// ---- BaseClasses/FB_CycleProfiler.TcPOU
// Core §8.11.4(b)/(f) — the cycle-time profile, fed by the step record the chain
// already keeps for §6.9: StepChanged() from _M_SetStep (with the step's time class,
// WORK by default), CycleComplete() at the finish step (§8.11.1 marker). Application
// steps add NOTHING except one enum on genuine wait steps. The step-chain / Unit
// base (M2) calls both automatically; until then a Unit wires the two calls once
// (Annex C §C.6). Fixed-size, no runtime allocation (Core §8.11.4(e)).
FUNCTION_BLOCK FB_CycleProfiler
VAR_OUTPUT
    Current        : ST_CycleProfile;   // cycle in progress (live waterfall)
    LastCycle      : ST_CycleProfile;   // last completed cycle — the HMI chart source
    StepStats      : ARRAY[1..PL_Fraktal.MAX_PROFILE_STEPS] OF ST_TimingRow;  // per-StepNo aggregates
    StatsTruncated : BOOL;
    // §8.11.1 throughput markers + §8.11.4 trend ring (the cycle-time ANALYSIS source:
    // per-cycle work/wait-class totals, charted by the HMI to explain increases)
    LastCycleTime  : TIME;
    MinCycleTime   : TIME;              // rolling minimum since reset (the demonstrated best)
    History        : ARRAY[1..PL_Fraktal.MAX_CYCLE_HISTORY] OF ST_CycleSummary;
    HistoryHead    : INT;               // newest entry (0 = none yet)
    // §8.11.4(d) — degradation is data: WorkTime drifting beyond Baseline*(1+BandPct)
    // pulses DegradedTrig for ONE call so the owner raises the maintenance event once.
    BaselineWorkMs : UDINT;             // 0 = degradation watch off (§3.8 config)
    DegradedBandPct: UDINT := 20;       // allowed drift above baseline, percent
    DegradedTrig   : BOOL;
    DegradedWorkMs : UDINT;             // the WorkTime that tripped the band (for the event text)
END_VAR
VAR
    _running      : BOOL;
    _openNo       : INT;
    _openName     : STRING(80);
    _openClass    : E_TimeClass;
    _openExpected : TIME;
    _openStartMs  : DWORD;
    _openStartDt  : DT;
    _openStartSynchronized : BOOL;
    _cycleStartMs : DWORD;
    _degraded     : BOOL;               // latched: one event per excursion, not per cycle
END_VAR

// no cyclic body — event-driven via StepChanged/CycleComplete

// fold the open step into the profile, the class split, and the aggregates
METHOD PRIVATE _M_CloseOpen
VAR_INPUT
    NowMs : DWORD;
END_VAR
VAR
    dur  : DWORD;
    i    : INT;
    slot : INT;
END_VAR
IF _openNo = 0 THEN
    RETURN;
END_IF
dur := NowMs - _openStartMs;                                // wrap-safe (TC3 §8.11)

// (1) ordered waterfall entry
IF Current.NSteps < PL_Fraktal.MAX_PROFILE_STEPS THEN
    Current.NSteps := Current.NSteps + 1;
    Current.Steps[Current.NSteps].StepNo   := _openNo;
    Current.Steps[Current.NSteps].StepName := _openName;
    Current.Steps[Current.NSteps].TimeClass:= _openClass;
    Current.Steps[Current.NSteps].Started  := _openStartDt;
    Current.Steps[Current.NSteps].StartedTimeSynchronized := _openStartSynchronized;
    Current.Steps[Current.NSteps].Duration := DWORD_TO_TIME(dur);
    Current.Steps[Current.NSteps].Expected := _openExpected;
ELSE
    Current.Truncated := TRUE;
END_IF

// (2) time-class split (§8.11.4(f)) — WorkTime/WaitTime derive from this at cycle close
Current.ByClass[TO_INT(_openClass)] := Current.ByClass[TO_INT(_openClass)] + DWORD_TO_TIME(dur);

// (3) per-StepNo aggregate (find-or-allocate; fixed array, Core §8.11.4(e))
slot := 0;
FOR i := 1 TO PL_Fraktal.MAX_PROFILE_STEPS DO
    IF (StepStats[i].Count > 0) AND (StepStats[i].Id = _openNo) THEN
        slot := i;
        EXIT;
    ELSIF (slot = 0) AND (StepStats[i].Count = 0) THEN
        slot := i;
    END_IF
END_FOR
IF slot = 0 THEN
    StatsTruncated := TRUE;
ELSE
    StepStats[slot].Id        := _openNo;
    StepStats[slot].Label     := _openName;
    StepStats[slot].TimeClass := _openClass;
    F_TimingUpdate(Row := StepStats[slot], DurMs := dur);
END_IF
END_METHOD

// §8.11.1 — discard the OPEN cycle without publishing it: a stop accepted at the
// between-cycles wait must not count a wait-only fragment as a production cycle
// (it would poison MinCycleTime and the trend). Aggregates keep completed cycles.
METHOD CycleAbandon : BOOL
_running := FALSE;
_openNo := 0;
CycleAbandon := TRUE;
END_METHOD

// close the open step and publish the cycle (call at the finish step, §8.11.1).
// Publishes WorkTime = ByClass[WORK] — the real cycle time (§8.11.4(f)).
METHOD CycleComplete : BOOL
VAR
    nowMs : DWORD;
END_VAR
IF NOT _running THEN
    CycleComplete := FALSE;
    RETURN;
END_IF
nowMs := TIME_TO_DWORD(TIME());
_M_CloseOpen(nowMs);
Current.Total    := DWORD_TO_TIME(nowMs - _cycleStartMs);   // wrap-safe (TC3 §8.11)
Current.WorkTime := Current.ByClass[TO_INT(E_TimeClass.WORK)];
Current.WaitTime := Current.Total - Current.WorkTime;
Current.CycleNo  := LastCycle.CycleNo + 1;
LastCycle := Current;

// §8.11.1 throughput markers
LastCycleTime := Current.Total;
IF (MinCycleTime = T#0S) OR (Current.Total < MinCycleTime) THEN
    MinCycleTime := Current.Total;
END_IF

// §8.11.4 trend ring — per-cycle class split for the HMI's cause analysis
HistoryHead := (HistoryHead MOD PL_Fraktal.MAX_CYCLE_HISTORY) + 1;
History[HistoryHead].CycleNo  := Current.CycleNo;
History[HistoryHead].Started  := Current.Started;
History[HistoryHead].StartedTimeSynchronized := Current.StartedTimeSynchronized;
History[HistoryHead].Total    := Current.Total;
History[HistoryHead].WorkTime := Current.WorkTime;
History[HistoryHead].WaitTime := Current.WaitTime;
History[HistoryHead].ByClass  := Current.ByClass;

// §8.11.4(d) — degradation watch on WORK time (waits are attributed, not drift).
// One-call trigger, latched per excursion; recovery below the band rearms it.
DegradedTrig := FALSE;
DegradedWorkMs := TIME_TO_DWORD(Current.WorkTime);
IF BaselineWorkMs > 0 THEN
    IF DegradedWorkMs * 100 > BaselineWorkMs * (100 + DegradedBandPct) THEN
        IF NOT _degraded THEN
            _degraded := TRUE;
            DegradedTrig := TRUE;
        END_IF
    ELSE
        _degraded := FALSE;
    END_IF
END_IF

_running := FALSE;
_openNo  := 0;
CycleComplete := TRUE;
END_METHOD

// Configure the recipe-owned WORK-time reference through the profiler owner.
// BaselineWorkMs is published read-only; TwinCAT therefore rejects assignment
// through a parent FB's published Profiler output. Zero disables the watch.
METHOD M_SetBaselineWork : BOOL
VAR_INPUT
    WorkMs : UDINT;
END_VAR
BaselineWorkMs := WorkMs;
DegradedTrig := FALSE;
_degraded := FALSE;
M_SetBaselineWork := TRUE;
END_METHOD

// deliberate, LOGGED action only (Core §8.11.2) — the caller raises the event
METHOD ResetStats : BOOL
VAR
    i     : INT;
    empty : ST_TimingRow;
    emptySummary : ST_CycleSummary;
END_VAR
FOR i := 1 TO PL_Fraktal.MAX_PROFILE_STEPS DO
    StepStats[i] := empty;
END_FOR
FOR i := 1 TO PL_Fraktal.MAX_CYCLE_HISTORY DO
    History[i] := emptySummary;
END_FOR
HistoryHead := 0;
LastCycleTime := T#0S;
MinCycleTime := T#0S;
_degraded := FALSE;
StatsTruncated := FALSE;
LastCycle.CycleNo := 0;
ResetStats := TRUE;
END_METHOD

// call on every step change — _M_SetStep already has StepNo/StepName (§6.5).
// TimeClass defaults to WORK; only genuine wait steps pass a wait class (§8.11.4(f)).
METHOD StepChanged : BOOL
VAR_INPUT
    StepNo   : INT;
    StepName : STRING(120);
    TimeClass    : E_TimeClass;
    Expected : TIME;                   // §8.11.4(c) — declared guard, drawn vs actual
END_VAR
VAR
    nowMs : DWORD;
    i     : INT;
END_VAR
IF _running AND (StepNo = _openNo) THEN
    _openClass := TimeClass;               // same step refreshed — class may be (re)declared
    _openExpected := Expected;
    StepChanged := TRUE;
    RETURN;
END_IF
nowMs := TIME_TO_DWORD(TIME());
IF NOT _running THEN
    _running := TRUE;                  // first step opens the cycle (§8.11.1 start marker)
    _cycleStartMs := nowMs;
    Current.Started   := F_Now();
    Current.StartedTimeSynchronized := F_TimeSynchronized();
    Current.NSteps    := 0;
    Current.Truncated := FALSE;
    FOR i := 0 TO 4 DO
        Current.ByClass[i] := T#0S;    // reset the class split for the new cycle
    END_FOR
ELSE
    _M_CloseOpen(nowMs);
END_IF
_openNo      := StepNo;
_openName    := StepName;
_openClass   := TimeClass;
_openExpected := Expected;
_openStartMs := nowMs;
_openStartDt := F_Now();
_openStartSynchronized := F_TimeSynchronized();
StepChanged := TRUE;
END_METHOD

END_FUNCTION_BLOCK

// ---- BaseClasses/FB_HostEventPublisher.TcPOU
// Core §11.6 — bounded per-Unit L3 event projection. Event production is local;
// transport is an optional injected sink and can never command the Unit.
FUNCTION_BLOCK FB_HostEventPublisher
VAR_OUTPUT
    Ring     : ARRAY[1..PL_Fraktal.MAX_HOST_EVENTS] OF ST_HostEvent;
    RingHead : INT;       // newest record, 0 when empty
    Count    : INT;       // valid records, saturates at the bound
    Capacity : INT := PL_Fraktal.MAX_HOST_EVENTS; // published bound; clients do not duplicate it
    Wrapped  : BOOL;      // oldest records have been overwritten
END_VAR
VAR
    {attribute 'OPC.UA.DA' := '0'}
    _sink : I_HostEventSink;
    _sequence : UDINT;
END_VAR

// event-driven; no cyclic body

METHOD Emit : BOOL
VAR_INPUT
    Kind          : E_HostEventKind;
    StationPath   : STRING(255);
    PartUid       : STRING(64);
    Subject       : STRING(80);
    Value         : STRING(80);
    Verdict       : E_Verdict;
    ReasonCode    : E_Reason;
END_VAR
VAR
    validKind : BOOL;
END_VAR
Emit := FALSE;
CASE Kind OF
    E_HostEventKind.PART_RECEIVED,
    E_HostEventKind.PROCESSING_STARTED,
    E_HostEventKind.PROCESSED,
    E_HostEventKind.PROCESSING_ABORTED,
    E_HostEventKind.CHANGEOVER_STARTED,
    E_HostEventKind.CHANGEOVER_DONE,
    E_HostEventKind.TOOL_CHANGED,
    E_HostEventKind.MATERIAL_CHANGED,
    E_HostEventKind.MODE_CHANGED,
    E_HostEventKind.NOK:
        validKind := TRUE;
ELSE
    validKind := FALSE;
END_CASE
IF NOT validKind OR (StationPath = '') THEN
    RETURN;
END_IF
_sequence := _sequence + 1;
RingHead := (RingHead MOD PL_Fraktal.MAX_HOST_EVENTS) + 1;
Ring[RingHead].Sequence := _sequence;
Ring[RingHead].Kind := Kind;
Ring[RingHead].StationPath := StationPath;
Ring[RingHead].PartUid := PartUid;
Ring[RingHead].Subject := Subject;
Ring[RingHead].Value := Value;
Ring[RingHead].Stamp := F_Now();
Ring[RingHead].TimeSynchronized := F_TimeSynchronized();
Ring[RingHead].Verdict := Verdict;
Ring[RingHead].ReasonCode := ReasonCode;
IF Count < PL_Fraktal.MAX_HOST_EVENTS THEN
    Count := Count + 1;
ELSE
    Wrapped := TRUE;
END_IF
IF _sink <> 0 THEN
    _sink.OnHostEvent(Ev := Ring[RingHead]);
END_IF
Emit := TRUE;
END_METHOD

METHOD SetSink : BOOL
VAR_INPUT
    Sink : I_HostEventSink;
END_VAR
_sink := Sink;
SetSink := TRUE;
END_METHOD

END_FUNCTION_BLOCK

// ---- Connectivity/FB_LineData.TcPOU
// Core §3.8e - data shared by every station on a line, held once. A line is NOT
// part of the Unit forest: it is no Unit, EM or CM, has no parent, and is never
// registered as anyone's child. The composition root declares it beside the roots
// (as it does a control domain, §9.8) and every root on the line references it
// with SetLine. A project registers its line values here (the ordinary
// M_RegisterConfig* calls, Kind := LINE_CFG, keys 'line.*'); each referencing
// root publishes them as its own line data and routes their writes here, so they
// are edited, audited and access-classed exactly like any other value, through
// the one mailbox. It extends FB_ModuleBase only because the typed value registry
// lives there (ModuleType NONE); commands are refused.
//
// The OWNER is the only editable copy; every accepted change raises Revision and
// the whole line is republished as Image. A MIRROR, on another controller or a
// root that is not the owner's, obtains the owner's Image through I_LineSource and
// applies a new revision whole or not at all; its values are read-only to every
// client. A mirror that stops updating keeps running on the revision it has and
// says so (Stale): a shift boundary one revision old is a reporting error, not a
// hazard, so staleness never blocks production on its own (§3.8e(d)).
FUNCTION_BLOCK FB_LineData EXTENDS FB_ModuleBase
VAR_INPUT
    ParCfg : ST_LineDataParCfg;
    ParCmd : ST_LineDataParCmd;
END_VAR
VAR_OUTPUT
    OutCmd : ST_LineDataOutCmd;
    OutImm : ST_LineStatus;       // §3.8e(d) - what this copy says about itself
    Image      : ST_LineImage;    // what a mirror reads, by symbol, over its source
END_VAR
VAR PERSISTENT
    _revision : UDINT;            // owner: current; mirror: last applied
    Calendar  : ST_ShiftCalendar; // §8.5.2 - line data like any other: edited at the owner
END_VAR
VAR
    {attribute 'OPC.UA.DA' := '0'}
    _source : I_LineSource;
    {attribute 'OPC.UA.DA' := '0'}
    _log : POINTER TO FB_AlarmLog;
    _role          : E_LineRole;
    _lastOkMs      : DWORD;
    _applied       : BOOL;        // not persistent: every boot re-applies once
    _imageBuilt    : BOOL;
    _imageRevision : UDINT;
    _syncing       : BOOL;
    _staleEvt      : INT;
    {attribute 'OPC.UA.DA' := '0'}
    _host          : PVOID;       // the root that ticks this line and lends its alarm log
    {attribute 'OPC.UA.DA' := '0'}
    _schedule : FB_ShiftSchedule;
    _dailyView : ST_ShiftCalendarV3;
    _incoming      : ST_LineImage; // mirror staging buffer - an instance member, never a local
END_VAR

Cyclic();

// OWNER takes no source. A MIRROR needs one, and StaleAfterMs is the window it
// declares for staying current (§3.8e(d)). Name is the line's own identity, never
// a path under a Unit.
METHOD Setup : BOOL
VAR_INPUT
    Name         : STRING(80);
    LineId       : STRING(40);
    Role         : E_LineRole;
    Source       : I_LineSource;
    StaleAfterMs : UDINT;
END_VAR
_M_SetName(Name);
Setup := FALSE;
IF (LineId = '') OR ((Role <> E_LineRole.OWNER) AND (Role <> E_LineRole.MIRROR)) THEN
    RETURN;
END_IF
IF (Role = E_LineRole.MIRROR) AND (Source = 0) THEN
    RETURN;                                // a mirror with nothing to mirror
END_IF
_role := Role;
_source := Source;
ParCfg.StaleAfterMs := StaleAfterMs;
OutImm.LineId := LineId;
OutImm.Role := Role;
IF (Role = E_LineRole.OWNER) AND (_revision = 0) THEN
    _revision := 1;                        // a published line is never at revision 0
END_IF
_lastOkMs := TIME_TO_DWORD(TIME());
Setup := _M_RegisterCalendar();
END_METHOD

// §8.5.2(a) - every line carries a shift calendar, registered identically on owner
// and mirror so a mirror can apply the owner's line whole.
METHOD PROTECTED _M_RegisterCalendar : BOOL
VAR
    n    : INT;
    ok   : BOOL;
    key  : STRING(160);
    item : STRING(255);
    label : STRING(160);
END_VAR
ok := M_RegisterConfigNumber(Key := 'line.shift.utcOffsetMin', Item := 'Calendar/UtcOffsetMin',
    LabelKey := 'std.config.shiftUtcOffset', Unit := E_EngUnit.MINUTE, Kind := E_ConfigKind.LINE_CFG,
    Storage := E_ConfigStorage.AS_DINT, pTarget := ADR(Calendar.UtcOffsetMin),
    Minimum := -720.0, Maximum := 840.0, RequiresReady := FALSE);
FOR n := 1 TO PL_Fraktal.MAX_SHIFTS DO
    key := CONCAT('line.shift.', CONCAT(TO_STRING(n), '.startMin'));
    item := CONCAT('Calendar/StartMin[', CONCAT(TO_STRING(n), ']'));
    // One label per shift: the four sit together in a root's line data group.
    label := CONCAT('std.config.shift.', CONCAT(TO_STRING(n), '.start'));
    ok := M_RegisterConfigNumber(Key := key, Item := item, LabelKey := label,
        Unit := E_EngUnit.MINUTE, Kind := E_ConfigKind.LINE_CFG, Storage := E_ConfigStorage.AS_DINT,
        pTarget := ADR(Calendar.StartMin[n]), Minimum := -1.0, Maximum := 1439.0,
        RequiresReady := FALSE) AND ok;
END_FOR
_M_RegisterCalendar := ok;
END_METHOD

// §3.8e(a) - called by FB_UnitBase.SetLine. The FIRST root to reference the line
// hosts it: it ticks the line once per scan and lends its alarm log for the
// staleness event. Every later root only references it; the host binding again
// stays the host. TRUE = you host it.
METHOD M_BindHost : BOOL
VAR_INPUT
    pHost     : PVOID;
    pAlarmLog : POINTER TO FB_AlarmLog;
END_VAR
M_BindHost := FALSE;
IF (pHost = 0) OR ((_host <> 0) AND (_host <> pHost)) THEN
    RETURN;
END_IF
_host := pHost;
_log := pAlarmLog;
M_BindHost := TRUE;
END_METHOD

// §3.8e - a referencing root publishes the line's values as ITS line data: under
// the root's scope, items prefixed 'Line/', keys 'line.*' (M_RegisterConfigWrite
// holds every line key to that prefix, so they cannot collide with the root's).
METHOD M_AppendLineConfig : BOOL
VAR_INPUT
    Pager : REFERENCE TO FB_ConfigPager;
    Scope : STRING(255);
END_VAR
_M_AppendCapabilities(Pager := Pager, Scope := Scope, ItemPrefix := 'Line/');
M_AppendLineConfig := TRUE;
END_METHOD

// §8.5.2 - minutes after LOCAL midnight for a UTC timestamp, with the line's offset.
METHOD M_MinuteOfDay : DINT
VAR_INPUT
    Now : DT;
END_VAR
VAR
    secOfDay : DINT;
END_VAR
secOfDay := UDINT_TO_DINT(DT_TO_UDINT(Now) MOD 86400) + Calendar.UtcOffsetMin * 60;
secOfDay := ((secOfDay MOD 86400) + 86400) MOD 86400;   // normalize a negative offset
M_MinuteOfDay := secOfDay / 60;
END_METHOD

// §8.5.2(a) - the used shift in force at a local minute: the latest start at or
// before it, and before the day's first start the day's LAST shift (a night shift
// wraps midnight). 0 when no shift is used. Complete by construction: no gaps.
METHOD M_CurrentShift : INT
VAR_INPUT
    MinuteOfDay : DINT;
END_VAR
VAR
    n           : INT;
    best        : INT;
    bestStart   : DINT;
    latest      : INT;
    latestStart : DINT;
END_VAR
best := 0;
bestStart := -1;
latest := 0;
latestStart := -1;
FOR n := 1 TO PL_Fraktal.MAX_SHIFTS DO
    IF (Calendar.StartMin[n] >= 0) AND (Calendar.StartMin[n] <= 1439) THEN
        IF (Calendar.StartMin[n] <= MinuteOfDay) AND (Calendar.StartMin[n] > bestStart) THEN
            best := n;
            bestStart := Calendar.StartMin[n];
        END_IF
        IF Calendar.StartMin[n] > latestStart THEN
            latest := n;
            latestStart := Calendar.StartMin[n];
        END_IF
    END_IF
END_FOR
IF best = 0 THEN
    best := latest;
END_IF
M_CurrentShift := best;
END_METHOD

METHOD PROTECTED OnCyclic : DINT
OnCyclic := SUPER^.OnCyclic();
CASE _role OF
    E_LineRole.OWNER:
        _M_BuildImage();
        OutImm.Owner := Status.Name;
        OutImm.Stale := FALSE;
    E_LineRole.MIRROR:
        _M_Mirror();
ELSE
    ;                                      // not set up: publishes nothing to mirror
END_CASE
OutImm.Revision := _revision;
END_METHOD

METHOD PROTECTED _M_Dispatch
_M_Fault(E_Reason.UNSUPPORTED_COMMAND, 'std.error.passiveInputHasNoCommand');
END_METHOD

METHOD PROTECTED _M_ConfigReadOnly : BOOL
_M_ConfigReadOnly := (_role = E_LineRole.MIRROR) AND NOT _syncing;
END_METHOD

// The owner's revision rises with every accepted change, so a mirror can tell a
// new line from the one it has. A mirror's own apply never counts.
METHOD M_ApplyConfigWrite : BOOL
VAR_INPUT
    Scope     : STRING(255);
    WriteKey  : STRING(160);
    Revision  : UDINT;
    TextValue : STRING(255);
    RootReady : BOOL;
END_VAR
M_ApplyConfigWrite := SUPER^.M_ApplyConfigWrite(Scope := Scope, WriteKey := WriteKey,
    Revision := Revision, TextValue := TextValue, RootReady := RootReady);
IF M_ApplyConfigWrite AND (_role = E_LineRole.OWNER) THEN
    _revision := _revision + 1;
END_IF
END_METHOD

// Republish the whole line when its revision moved (or on the first scan, after
// every value has been registered). Values change only through the write path.
METHOD PRIVATE _M_BuildImage
VAR
    i     : INT;
    count : INT;
END_VAR
IF _imageBuilt AND (_imageRevision = _revision) THEN
    RETURN;
END_IF
Image.LineId := OutImm.LineId;
Image.Owner := Status.Name;
Image.Revision := _revision;
count := 0;
FOR i := 1 TO _nConfigWrite DO
    IF (_pConfigWrite[i - 1].Kind = E_ConfigKind.LINE_CFG)
    AND (count < PL_Fraktal.MAX_LINE_RECORDS) THEN
        count := count + 1;
        Image.Records[count].WriteKey := _pConfigWrite[i - 1].Key;
        Image.Records[count].Revision := _pConfigWrite[i - 1].Revision;
        Image.Records[count].ValueText := _M_ConfigValueText(Idx := i);
    END_IF
END_FOR
Image.Count := count;
_imageRevision := _revision;
_imageBuilt := TRUE;
END_METHOD

METHOD PRIVATE _M_Mirror
VAR
    ok      : BOOL;
    nowMs   : DWORD;
    elapsed : DWORD;
END_VAR
ok := FALSE;
nowMs := TIME_TO_DWORD(TIME());
IF _source.M_Poll(Image := _incoming) THEN
    IF _incoming.LineId <> OutImm.LineId THEN
        OutImm.SourceError := 1;       // somebody else's line: never applied
    ELSIF _applied AND (_incoming.Revision = _revision) THEN
        ok := TRUE;                        // current
    ELSIF _M_ApplyIncoming() THEN
        _revision := _incoming.Revision;
        _applied := TRUE;
        Image := _incoming;
        OutImm.Owner := _incoming.Owner;
        ok := TRUE;
    ELSE
        OutImm.SourceError := 2;       // not applicable whole: nothing applied
    END_IF
ELSIF _source.M_Error() <> 0 THEN
    OutImm.SourceError := _source.M_Error();
END_IF
IF ok THEN
    _lastOkMs := nowMs;
    OutImm.SourceError := 0;
    OutImm.LastUpdate := F_Now();
    OutImm.TimeSynchronized := F_TimeSynchronized();
END_IF
// Unsigned subtraction: a wrapping millisecond counter never fakes an expiry.
elapsed := nowMs - _lastOkMs;
OutImm.Stale := elapsed > TO_DWORD(ParCfg.StaleAfterMs);
IF OutImm.Stale AND (_staleEvt = 0) AND (_log <> 0) THEN
    _staleEvt := _log^.Raise(Reason := E_Reason.NONE, Text := 'std.error.lineDataStale',
        Source := Status.Name, Severity := E_Severity.LOW, Category := E_Category.SYSTEM,
        ResetClass := E_ResetClass.AUTO_RESET);
ELSIF NOT OutImm.Stale AND (_staleEvt > 0) THEN
    IF _log <> 0 THEN
        _log^.Gone(Slot := _staleEvt);
    END_IF
    _staleEvt := 0;
END_IF
END_METHOD

// §3.8e(c) - whole or not at all. The image must carry exactly the line values
// this copy registered; every record is staged through its typed handler before
// any is applied, as a §3.8b set load is.
METHOD PRIVATE _M_ApplyIncoming : BOOL
VAR
    i     : INT;
    j     : INT;
    n     : INT;
    local : INT;
END_VAR
_M_ApplyIncoming := FALSE;
n := LIMIT(0, _incoming.Count, PL_Fraktal.MAX_LINE_RECORDS);
local := 0;
FOR i := 1 TO _nConfigWrite DO
    IF _pConfigWrite[i - 1].Kind = E_ConfigKind.LINE_CFG THEN
        local := local + 1;
    END_IF
END_FOR
IF (n <> local) OR (n <> _incoming.Count) THEN
    RETURN;                                // the two sides disagree on what the line is
END_IF
// Duplicate identities cannot substitute for a missing field.
FOR i := 1 TO n DO
    FOR j := i + 1 TO n DO
        IF _incoming.Records[i].WriteKey = _incoming.Records[j].WriteKey THEN RETURN; END_IF
    END_FOR
END_FOR
IF NOT M_BeginConfigBatch() THEN RETURN; END_IF
_syncing := TRUE;
FOR i := 1 TO n DO
    IF NOT M_StageConfigWrite(Scope := Status.Name, WriteKey := _incoming.Records[i].WriteKey,
            Revision := _incoming.Records[i].Revision,
            TextValue := _incoming.Records[i].ValueText, RootReady := TRUE) THEN
        M_EndConfigBatch();
        _syncing := FALSE;
        RETURN;
    END_IF
END_FOR
IF NOT M_ValidateConfigBatch() THEN
    M_EndConfigBatch(); _syncing := FALSE; RETURN;
END_IF
FOR i := 1 TO n DO
    M_ApplyConfigWrite(Scope := Status.Name, WriteKey := _incoming.Records[i].WriteKey,
        Revision := _incoming.Records[i].Revision,
        TextValue := _incoming.Records[i].ValueText, RootReady := TRUE);
END_FOR
M_CommitConfigBatch();
_syncing := FALSE;
_M_ApplyIncoming := TRUE;
END_METHOD

METHOD M_ShiftInterval : BOOL
VAR_INPUT
    Now : DT;
END_VAR
VAR_OUTPUT
    ShiftIndex : INT;
    StartAt : DT;
    EndAt : DT;
    Target : UDINT;
END_VAR
M_ShiftInterval := _schedule.M_MigrateV1(Source := Calendar, Target := _dailyView);
IF M_ShiftInterval THEN
    _schedule.M_Interval(Now := Now, Calendar := _dailyView,
        ShiftIndex => ShiftIndex, StartAt => StartAt, EndAt => EndAt, Target => Target);
END_IF
END_METHOD

METHOD M_BeginConfigBatch : BOOL
M_BeginConfigBatch := TRUE;
END_METHOD

METHOD M_ValidateConfigBatch : BOOL
M_ValidateConfigBatch := TRUE;
END_METHOD

METHOD M_EndConfigBatch
;
END_METHOD

METHOD M_CommitConfigBatch : BOOL
M_CommitConfigBatch := TRUE;
END_METHOD

END_FUNCTION_BLOCK

// ---- Connectivity/FB_ShiftSchedule.TcPOU
FUNCTION_BLOCK FB_ShiftSchedule

;

// Half-open weekly intervals, including Sunday-to-Monday wrap.
METHOD M_Validate : BOOL
VAR_IN_OUT
    Calendar : ST_ShiftCalendarV3;
END_VAR
VAR
    i, j, dayI, dayJ, delta : INT;
    startI, endI, startJ, endJ : DINT;
END_VAR
M_Validate := FALSE;
IF (Calendar.SchemaVersion <> 3) OR (Calendar.UtcOffsetMin < -840)
OR (Calendar.UtcOffsetMin > 840) THEN RETURN; END_IF
FOR i := 1 TO PL_Fraktal.MAX_WEEKLY_SHIFTS DO
    IF (Calendar.Rows[i].StartMin < -1) OR (Calendar.Rows[i].StartMin > 1439)
    OR (Calendar.Rows[i].DurationMin < 1) OR (Calendar.Rows[i].DurationMin > 1440)
    OR (Calendar.Rows[i].ActiveDays < 0) OR (Calendar.Rows[i].ActiveDays > 127)
    OR (Calendar.Rows[i].ProductionTarget < 0) THEN RETURN; END_IF
END_FOR
FOR i := 1 TO PL_Fraktal.MAX_WEEKLY_SHIFTS DO
    IF Calendar.Rows[i].StartMin >= 0 THEN
        FOR dayI := 0 TO 6 DO
            IF (TO_DWORD(Calendar.Rows[i].ActiveDays) AND SHL(DWORD#1, dayI)) <> 0 THEN
                startI := dayI * 1440 + Calendar.Rows[i].StartMin;
                endI := startI + Calendar.Rows[i].DurationMin;
                FOR j := i TO PL_Fraktal.MAX_WEEKLY_SHIFTS DO
                    IF Calendar.Rows[j].StartMin >= 0 THEN
                        FOR dayJ := 0 TO 6 DO
                            IF ((j <> i) OR (dayJ <> dayI))
                            AND ((TO_DWORD(Calendar.Rows[j].ActiveDays) AND SHL(DWORD#1, dayJ)) <> 0) THEN
                                FOR delta := -1 TO 1 DO
                                    startJ := dayJ * 1440 + Calendar.Rows[j].StartMin + delta * 10080;
                                    endJ := startJ + Calendar.Rows[j].DurationMin;
                                    IF (startI < endJ) AND (startJ < endI) THEN RETURN; END_IF
                                END_FOR
                            END_IF
                        END_FOR
                    END_IF
                END_FOR
            END_IF
        END_FOR
    END_IF
END_FOR
M_Validate := TRUE;
END_METHOD

// Called at interval entry/boundary, not on every production scan.
METHOD M_Interval : BOOL
VAR_INPUT
    Now : DT;
END_VAR
VAR_IN_OUT
    Calendar : ST_ShiftCalendarV3;
END_VAR
VAR_OUTPUT
    ShiftIndex : INT;
    StartAt : DT;
    EndAt : DT; // zero means no finite next boundary
    Target : UDINT;
END_VAR
VAR
    nowSec, localSec, weekStart, startSec, endSec, nextSec : LINT;
    dayNo : LINT;
    i, day, week : INT;
END_VAR
M_Interval := TRUE;
ShiftIndex := 0; StartAt := Now; EndAt := DT#1970-01-01-00:00:00; Target := 0;
nowSec := TO_LINT(DT_TO_UDINT(Now));
localSec := nowSec + Calendar.UtcOffsetMin * LINT#60;
dayNo := localSec / 86400;
IF localSec < 0 THEN dayNo := (localSec - 86399) / 86400; END_IF
weekStart := (dayNo - ((dayNo + 3 + 7) MOD 7)) * 86400;
nextSec := LINT#4294967296;
FOR i := 1 TO PL_Fraktal.MAX_WEEKLY_SHIFTS DO
    IF (Calendar.Rows[i].StartMin >= 0) AND (Calendar.Rows[i].ActiveDays > 0) THEN
        FOR day := 0 TO 6 DO
            IF (TO_DWORD(Calendar.Rows[i].ActiveDays) AND SHL(DWORD#1, day)) <> 0 THEN
                FOR week := -1 TO 1 DO
                    startSec := weekStart + week * LINT#604800 + day * LINT#86400
                        + Calendar.Rows[i].StartMin * LINT#60 - Calendar.UtcOffsetMin * LINT#60;
                    endSec := startSec + Calendar.Rows[i].DurationMin * LINT#60;
                    IF (startSec <= nowSec) AND (nowSec < endSec) THEN
                        ShiftIndex := i;
                        IF startSec >= 0 THEN StartAt := UDINT_TO_DT(TO_UDINT(startSec)); END_IF
                        IF endSec <= 4294967295 THEN EndAt := UDINT_TO_DT(TO_UDINT(endSec)); END_IF
                        Target := TO_UDINT(Calendar.Rows[i].ProductionTarget);
                    END_IF
                    IF (startSec > nowSec) AND (startSec < nextSec) THEN nextSec := startSec; END_IF
                END_FOR
            END_IF
        END_FOR
    END_IF
END_FOR
IF (ShiftIndex = 0) AND (nextSec <= 4294967295) THEN EndAt := UDINT_TO_DT(TO_UDINT(nextSec)); END_IF
END_METHOD

METHOD M_MigrateV1 : BOOL
VAR_IN_OUT
    Source : ST_ShiftCalendar;
    Target : ST_ShiftCalendarV3;
END_VAR
VAR
    i, j : INT;
    duration, distance : DINT;
END_VAR
M_MigrateV1 := FALSE;
Target.SchemaVersion := 3;
Target.UtcOffsetMin := Source.UtcOffsetMin;
FOR i := 1 TO PL_Fraktal.MAX_WEEKLY_SHIFTS DO
    Target.Rows[i].StartMin := -1;
    Target.Rows[i].DurationMin := 1440;
    Target.Rows[i].ActiveDays := 0;
    Target.Rows[i].ProductionTarget := 0;
END_FOR
FOR i := 1 TO PL_Fraktal.MAX_SHIFTS DO
    IF (Source.StartMin[i] < -1) OR (Source.StartMin[i] > 1439) THEN RETURN; END_IF
    IF Source.StartMin[i] >= 0 THEN
        duration := 1440;
        FOR j := 1 TO PL_Fraktal.MAX_SHIFTS DO
            IF (j <> i) AND (Source.StartMin[j] >= 0) THEN
                distance := (Source.StartMin[j] - Source.StartMin[i] + 1440) MOD 1440;
                IF distance = 0 THEN RETURN; END_IF
                IF distance < duration THEN duration := distance; END_IF
            END_IF
        END_FOR
        Target.Rows[i].StartMin := Source.StartMin[i];
        Target.Rows[i].DurationMin := duration;
        Target.Rows[i].ActiveDays := 127;
    END_IF
END_FOR
M_MigrateV1 := M_Validate(Calendar := Target);
END_METHOD

METHOD M_MigrateV2 : BOOL
VAR_IN_OUT
    Source : ST_ShiftCalendarV2;
    Target : ST_ShiftCalendarV3;
END_VAR
VAR
    i : INT;
END_VAR
M_MigrateV2 := FALSE;
IF Source.SchemaVersion <> 2 THEN RETURN; END_IF
Target.SchemaVersion := 3;
Target.UtcOffsetMin := Source.UtcOffsetMin;
FOR i := 1 TO PL_Fraktal.MAX_WEEKLY_SHIFTS DO
    Target.Rows[i].StartMin := -1;
    Target.Rows[i].DurationMin := 1440;
    Target.Rows[i].ActiveDays := 0;
    Target.Rows[i].ProductionTarget := 0;
END_FOR
FOR i := 1 TO PL_Fraktal.MAX_SHIFTS DO
    Target.Rows[i].StartMin := Source.Rows[i].StartMin;
    Target.Rows[i].DurationMin := Source.Rows[i].DurationMin;
    Target.Rows[i].ActiveDays := Source.Rows[i].ActiveDays;
END_FOR
M_MigrateV2 := M_Validate(Calendar := Target);
END_METHOD

END_FUNCTION_BLOCK

// ---- BaseClasses/FB_SystemHealthPublisher.TcPOU
// Core §2.7/§8.12 — one bounded, reusable health evaluator. Platform adapters
// supply measurements; this owner publishes live values and owns alarm edges.
FUNCTION_BLOCK FB_SystemHealthPublisher
VAR_OUTPUT
    Status : ST_SystemHealthStatus;
END_VAR
VAR
    {attribute 'OPC.UA.DA' := '0'}
    _log : POINTER TO FB_AlarmLog;
    _sourcePath : STRING(255);
    _taskOverrunSlot, _taskJitterSlot, _controllerSlot : INT;
    _cpuSlot, _memorySlot, _temperatureSlot, _fanSlot, _storageSlot : INT;
    _fieldbusSlot, _dcSlot, _timeSlot : INT;
END_VAR

;

METHOD Setup : BOOL
VAR_INPUT
    SourcePath : STRING(255);
    pAlarmLog  : POINTER TO FB_AlarmLog;
END_VAR
_sourcePath := SourcePath;
_log := pAlarmLog;
Status.SourcePath := SourcePath;
Setup := (_sourcePath <> '') AND (_log <> 0);
END_METHOD

METHOD Cyclic : BOOL
VAR_INPUT
    Input      : ST_SystemHealthInput;
    ParCfg     : ST_SystemHealthParCfg;
    Configured : BOOL;
END_VAR
VAR
    validCfg, taskOverrunBad, jitterBad, controllerBad : BOOL;
    cpuBad, memoryBad, temperatureBad, fanBad, storageBad : BOOL;
    fieldbusBad, dcBad, timeBad : BOOL;
END_VAR
validCfg := Configured AND (ParCfg.SchemaVersion = 1)
    AND (ParCfg.MaxTaskCycleUs > 0) AND (ParCfg.MaxTaskJitterUs > 0)
    AND (ParCfg.MaxCpuLoadPct > 0.0) AND (ParCfg.MaxCpuLoadPct <= 100.0)
    AND (ParCfg.MaxIpcTemperatureC > 0.0)
    AND (ParCfg.MinStorageHealthPct >= 0.0) AND (ParCfg.MinStorageHealthPct <= 100.0)
    AND (ParCfg.MaxTimeOffsetUs >= 0);

Status.Present := validCfg;
Status.SourcePath := _sourcePath;
Status.TaskAvailable := Input.TaskAvailable;
Status.TaskCycleUs := Input.TaskCycleUs;
Status.TaskJitterUs := Input.TaskJitterUs;
Status.TaskOverrun := Input.TaskOverrun;
Status.ControllerAvailable := Input.ControllerAvailable;
Status.CpuLoadPct := Input.CpuLoadPct;
Status.MemoryAvailableMb := Input.MemoryAvailableMb;
Status.IpcAvailable := Input.IpcAvailable;
Status.IpcTemperatureC := Input.IpcTemperatureC;
Status.FanHealthy := Input.FanHealthy;
Status.StorageHealthPct := Input.StorageHealthPct;
Status.FieldbusAvailable := Input.FieldbusAvailable;
Status.FieldbusMasterHealthy := Input.FieldbusMasterHealthy;
Status.LostFrameCount := Input.LostFrameCount;
Status.SlaveErrorCount := Input.SlaveErrorCount;
Status.DcAvailable := Input.DcAvailable;
Status.DcSynchronized := Input.DcSynchronized;
Status.TimeQuality := Input.TimeQuality;
Status.FanAvailable := Input.IpcAvailable AND Input.FanAvailable;
Status.StorageAvailable := Input.IpcAvailable AND Input.StorageAvailable;

taskOverrunBad := validCfg AND (NOT Input.TaskAvailable OR Input.TaskOverrun
    OR (Input.TaskCycleUs > ParCfg.MaxTaskCycleUs));
jitterBad := validCfg AND Input.TaskAvailable
    AND (Input.TaskJitterUs > ParCfg.MaxTaskJitterUs);
controllerBad := validCfg AND NOT Input.ControllerAvailable;
cpuBad := validCfg AND Input.ControllerAvailable
    AND (Input.CpuLoadPct > ParCfg.MaxCpuLoadPct);
memoryBad := validCfg AND Input.ControllerAvailable
    AND (Input.MemoryAvailableMb < ParCfg.MinMemoryAvailableMb);
temperatureBad := validCfg AND Input.IpcAvailable
    AND (Input.IpcTemperatureC > ParCfg.MaxIpcTemperatureC);
fanBad := validCfg AND Input.IpcAvailable AND Input.FanAvailable
    AND NOT Input.FanHealthy;
storageBad := validCfg AND Input.IpcAvailable AND Input.StorageAvailable
    AND (Input.StorageHealthPct < ParCfg.MinStorageHealthPct);
fieldbusBad := validCfg AND (Input.FieldbusAvailable
    AND (NOT Input.FieldbusMasterHealthy
        OR (Input.LostFrameCount > ParCfg.MaxLostFrames)
        OR (Input.SlaveErrorCount > ParCfg.MaxSlaveErrors))
    OR (ParCfg.RequireFieldbus AND NOT Input.FieldbusAvailable));
dcBad := validCfg AND ParCfg.RequireDcSync
    AND (NOT Input.DcAvailable OR NOT Input.DcSynchronized);
timeBad := validCfg AND ParCfg.RequireTimeSync
    AND (NOT Input.TimeQuality.Available OR NOT Input.TimeQuality.Synchronized
        OR (Input.TimeQuality.OffsetUs > ParCfg.MaxTimeOffsetUs)
        OR (Input.TimeQuality.OffsetUs < -ParCfg.MaxTimeOffsetUs));

_M_UpdateAlarm(Active := taskOverrunBad, Reason := E_Reason.TASK_OVERRUN,
    Text := 'std.system.taskOverrun', Slot := _taskOverrunSlot);
_M_UpdateAlarm(Active := jitterBad, Reason := E_Reason.TASK_JITTER_HIGH,
    Text := 'std.system.taskJitterHigh', Slot := _taskJitterSlot);
_M_UpdateAlarm(Active := controllerBad, Reason := E_Reason.CONTROLLER_METRICS_UNAVAILABLE,
    Text := 'std.system.controllerMetricsUnavailable', Slot := _controllerSlot);
_M_UpdateAlarm(Active := cpuBad, Reason := E_Reason.CPU_LOAD_HIGH,
    Text := 'std.system.cpuLoadHigh', Slot := _cpuSlot);
_M_UpdateAlarm(Active := memoryBad, Reason := E_Reason.MEMORY_LOW,
    Text := 'std.system.memoryLow', Slot := _memorySlot);
_M_UpdateAlarm(Active := temperatureBad, Reason := E_Reason.IPC_TEMP_HIGH,
    Text := 'std.system.ipcTemperatureHigh', Slot := _temperatureSlot);
_M_UpdateAlarm(Active := fanBad, Reason := E_Reason.IPC_FAN_FAULT,
    Text := 'std.system.ipcFanFault', Slot := _fanSlot);
_M_UpdateAlarm(Active := storageBad, Reason := E_Reason.STORAGE_HEALTH_LOW,
    Text := 'std.system.storageHealthLow', Slot := _storageSlot);
_M_UpdateAlarm(Active := fieldbusBad, Reason := E_Reason.FIELDBUS_MASTER_FAULT,
    Text := 'std.system.fieldbusMasterFault', Slot := _fieldbusSlot);
_M_UpdateAlarm(Active := dcBad, Reason := E_Reason.DC_SYNC_LOST,
    Text := 'std.system.dcSyncLost', Slot := _dcSlot);
_M_UpdateAlarm(Active := timeBad, Reason := E_Reason.TIME_SYNC_LOST,
    Text := 'std.system.timeSyncLost', Slot := _timeSlot);

Status.Healthy := validCfg AND NOT taskOverrunBad AND NOT jitterBad
    AND NOT controllerBad AND NOT cpuBad AND NOT memoryBad
    AND NOT temperatureBad AND NOT fanBad AND NOT storageBad
    AND NOT fieldbusBad AND NOT dcBad AND NOT timeBad;
Cyclic := validCfg;
END_METHOD

METHOD PRIVATE _M_UpdateAlarm
VAR_INPUT
    Active : BOOL;
    Reason : E_Reason;
    Text   : STRING(255);
END_VAR
VAR_IN_OUT
    Slot : INT;
END_VAR
IF Active THEN
    IF (Slot = 0) AND (_log <> 0) THEN
        Slot := _log^.Raise(Reason := Reason, Text := Text, Source := _sourcePath,
            Severity := E_Severity.LOW, Category := E_Category.SYSTEM,
            ResetClass := E_ResetClass.AUTO_RESET);
    END_IF
ELSE
    IF (Slot > 0) AND (_log <> 0) THEN
        _log^.Gone(Slot := Slot);
    END_IF
    Slot := 0;
END_IF
END_METHOD

END_FUNCTION_BLOCK

// ---- BaseClasses/FB_SignalTower.TcPOU
// Core §8.13 — single state/alarm/operator-action mapping plus bounded lamp test.
// Outputs are semantics only; the project Hardware Driver owns electrical I/O.
FUNCTION_BLOCK FB_SignalTower
VAR_OUTPUT
    Status : ST_SignalTowerOut;
END_VAR
VAR
    _testEdge : R_TRIG;
    _testTimer : TON;
    _testActive : BOOL;
END_VAR

;

METHOD Cyclic : BOOL
VAR_INPUT
    MachineState          : E_MachineState;
    AlarmActive           : BOOL;
    HighestSeverity       : E_Severity;
    OperatorActionRequired: BOOL;
    LampTestRequest       : BOOL;
    ParCfg                : ST_SignalTowerParCfg;
END_VAR
VAR
    duration : TIME;
END_VAR
duration := ParCfg.LampTestDuration;
IF (ParCfg.SchemaVersion <> 1) OR (duration <= T#0S) THEN
    duration := T#3S;
ELSIF duration > T#30S THEN
    duration := T#30S;
ELSE
    ;
END_IF
_testEdge(CLK := LampTestRequest);
IF _testEdge.Q THEN
    _testActive := TRUE;
    _testTimer(IN := FALSE);
END_IF
_testTimer(IN := _testActive, PT := duration);
IF _testTimer.Q THEN
    _testActive := FALSE;
    _testTimer(IN := FALSE);
END_IF

Status.Red := FALSE;
Status.Amber := FALSE;
Status.Green := FALSE;
Status.Blue := FALSE;
Status.White := FALSE;
Status.Horn := FALSE;
Status.TestActive := _testActive;
IF _testActive THEN
    Status.Red := TRUE;
    Status.Amber := TRUE;
    Status.Green := TRUE;
    Status.Blue := TRUE;
    Status.White := TRUE;
    Status.Horn := TRUE;
ELSE
    CASE MachineState OF
        E_MachineState.DOWN:
            Status.Red := TRUE;
        E_MachineState.BLOCKED, E_MachineState.STARVED, E_MachineState.CHANGEOVER:
            Status.Amber := TRUE;
        E_MachineState.PRODUCING:
            Status.Green := TRUE;
        E_MachineState.IDLE, E_MachineState.STOPPED:
            ;
        ELSE
            Status.Red := TRUE; // unknown state fails conspicuously
    END_CASE
    IF AlarmActive THEN
        CASE HighestSeverity OF
            E_Severity.HIGH:
                Status.Red := TRUE;
                Status.Green := FALSE;
                IF ParCfg.HornOnHigh THEN Status.Horn := TRUE; ELSE ; END_IF
            E_Severity.MED, E_Severity.LOW:
                IF NOT Status.Red THEN Status.Amber := TRUE; ELSE ; END_IF
            ELSE
                Status.Red := TRUE;
                Status.Green := FALSE;
        END_CASE
    ELSE
        ;
    END_IF
    IF OperatorActionRequired THEN
        IF ParCfg.OperatorUsesWhite THEN Status.White := TRUE; ELSE Status.Blue := TRUE; END_IF
    ELSE
        ;
    END_IF
END_IF
Cyclic := TRUE;
END_METHOD

END_FUNCTION_BLOCK

// ---- Platform/F_ManualEnable.TcPOU
// Core §9 — derive the manual-enable fact from the published safety devices.
// Pure, bounded, and fail-closed: no enabling device mirrored means NOT held,
// so a cell that never wired one cannot jog with its guards open by omission.
//
// Grepping for calls to this function lists every place in a codebase where
// motion is authorised by an enabling device. That auditability is the point of
// deriving it here rather than letting each station assemble the condition.
FUNCTION F_ManualEnable : ST_ManualEnableStatus
VAR_INPUT
    Safety : ST_SafetyStatus;
END_VAR
VAR
    i : INT;
END_VAR

// Fail-closed defaults (§5.6, O10): every early return leaves Held FALSE.
F_ManualEnable.Present    := FALSE;
F_ManualEnable.Held       := FALSE;
F_ManualEnable.DeviceName := '';

IF NOT Safety.Present THEN
    RETURN;                       // no safety facet at all -> nothing to permit with
END_IF

FOR i := 1 TO PL_Fraktal.MAX_SAFETY_DEVICES DO
    IF Safety.Devices[i].Present AND (Safety.Devices[i].Kind = E_SafetyDeviceKind.ENABLE_SWITCH) THEN
        F_ManualEnable.Present := TRUE;
        // Permitting is the POSITIVE state, exactly as an E-stop that is not
        // pressed publishes Ready/NOT DemandActive (§9). A released or
        // panic-squeezed enabling device demands the safe state like any other
        // device, so it fails every one of these tests.
        IF Safety.Devices[i].Ready
            AND NOT Safety.Devices[i].DemandActive
            AND NOT Safety.Devices[i].SafeStateActive
            AND NOT Safety.Devices[i].FaultActive
            AND Safety.Devices[i].FieldbusHealthy
            AND (Safety.Devices[i].State = E_SafetyState.READY)
            // A fault anywhere in the facet withdraws the permission even while
            // this device reads as held: a safety system reporting a fault is
            // not one to take permission from (O10). It must be tested HERE -
            // a check after the loop never ran, because a held device RETURNs.
            AND NOT Safety.FaultActive THEN
            F_ManualEnable.Held       := TRUE;
            F_ManualEnable.DeviceName := Safety.Devices[i].Name;
            RETURN;                   // first permitting device wins and names itself
        END_IF
    END_IF
END_FOR

END_FUNCTION

// ---- Connectivity/FB_LineDataV3.TcPOU
// Versioned weekly Line owner/mirror; inherited V1 image is retained for migration.
FUNCTION_BLOCK FB_LineDataV3 EXTENDS FB_LineData
VAR PERSISTENT
    CalendarV2 : ST_ShiftCalendarV2; // explicit V2 migration image, never reinterpreted
    CalendarV3 : ST_ShiftCalendarV3;
END_VAR
VAR
    {attribute 'OPC.UA.DA' := '0'}
    _weeklyConfig : ARRAY[1..21] OF ST_ConfigWriteDef;
    _candidate : ST_ShiftCalendarV3;
    _batch : BOOL;
END_VAR

Cyclic();

METHOD PROTECTED _M_RegisterCalendar : BOOL
VAR
    n : INT;
    ok : BOOL;
    found : UINT;
    key : STRING(160);
    item : STRING(255);
    label : STRING(160);
END_VAR
_M_RegisterCalendar := FALSE;
IF NOT _M_UseConfigRegistry(pRecords := ADR(_weeklyConfig), Capacity := 21) THEN RETURN; END_IF
IF CalendarV3.SchemaVersion = 0 THEN
    IF CalendarV2.SchemaVersion = 2 THEN
        ok := _schedule.M_MigrateV2(Source := CalendarV2, Target := _candidate);
    ELSIF CalendarV2.SchemaVersion = 0 THEN
        ok := _schedule.M_MigrateV1(Source := Calendar, Target := _candidate);
    ELSE
        // A present incompatible weekly image is not a missing image.
        ok := FALSE;
    END_IF
    IF ok THEN CalendarV3 := _candidate; END_IF
END_IF
IF NOT _schedule.M_Validate(Calendar := CalendarV3) THEN
    // Reject a real incompatible image visibly; keep the schedule empty.
    found := CalendarV3.SchemaVersion;
    IF found = 0 THEN found := 65535; END_IF
    M_RestoreStationCfg(pVersion := ADR(found), SchemaVersion := 3);
    CalendarV3.SchemaVersion := 3;
    CalendarV3.UtcOffsetMin := 0;
    FOR n := 1 TO PL_Fraktal.MAX_WEEKLY_SHIFTS DO
        CalendarV3.Rows[n].StartMin := -1;
        CalendarV3.Rows[n].DurationMin := 1440;
        CalendarV3.Rows[n].ActiveDays := 0;
        CalendarV3.Rows[n].ProductionTarget := 0;
    END_FOR
END_IF
ok := M_RegisterConfigNumber(Key := 'line.shift.utcOffsetMin', Item := 'CalendarV3/UtcOffsetMin',
    LabelKey := 'std.config.shiftUtcOffset', Unit := E_EngUnit.MINUTE, Kind := E_ConfigKind.LINE_CFG,
    Storage := E_ConfigStorage.AS_DINT, pTarget := ADR(CalendarV3.UtcOffsetMin),
    Minimum := -840.0, Maximum := 840.0, RequiresReady := FALSE);
M_SetConfigAccess(WriteKey := 'line.shift.utcOffsetMin', ClassId := '',
    MinReadLevel := E_AccessLevel.NONE, MinWriteLevel := E_AccessLevel.ENGINEER);
FOR n := 1 TO PL_Fraktal.MAX_WEEKLY_SHIFTS DO
    key := CONCAT('line.shift.', CONCAT(TO_STRING(n), '.startMin'));
    item := CONCAT('CalendarV3/Rows[', CONCAT(TO_STRING(n), ']/StartMin'));
    label := CONCAT('std.config.shift.', CONCAT(TO_STRING(n), '.start'));
    ok := M_RegisterConfigNumber(Key := key, Item := item, LabelKey := label,
        Unit := E_EngUnit.MINUTE, Kind := E_ConfigKind.LINE_CFG, Storage := E_ConfigStorage.AS_DINT,
        pTarget := ADR(CalendarV3.Rows[n].StartMin), Minimum := -1.0, Maximum := 1439.0,
        RequiresReady := FALSE) AND ok;
    M_SetConfigAccess(WriteKey := key, ClassId := '', MinReadLevel := E_AccessLevel.NONE,
        MinWriteLevel := E_AccessLevel.ENGINEER);
    key := CONCAT('line.shift.', CONCAT(TO_STRING(n), '.durationMin'));
    item := CONCAT('CalendarV3/Rows[', CONCAT(TO_STRING(n), ']/DurationMin'));
    label := CONCAT('std.config.shift.', CONCAT(TO_STRING(n), '.duration'));
    ok := M_RegisterConfigNumber(Key := key, Item := item, LabelKey := label,
        Unit := E_EngUnit.MINUTE, Kind := E_ConfigKind.LINE_CFG, Storage := E_ConfigStorage.AS_DINT,
        pTarget := ADR(CalendarV3.Rows[n].DurationMin), Minimum := 1.0, Maximum := 1440.0,
        RequiresReady := FALSE) AND ok;
    M_SetConfigAccess(WriteKey := key, ClassId := '', MinReadLevel := E_AccessLevel.NONE,
        MinWriteLevel := E_AccessLevel.ENGINEER);
    key := CONCAT('line.shift.', CONCAT(TO_STRING(n), '.activeDays'));
    item := CONCAT('CalendarV3/Rows[', CONCAT(TO_STRING(n), ']/ActiveDays'));
    label := CONCAT('std.config.shift.', CONCAT(TO_STRING(n), '.activeDays'));
    ok := M_RegisterConfigNumber(Key := key, Item := item, LabelKey := label,
        Unit := E_EngUnit.NONE, Kind := E_ConfigKind.LINE_CFG, Storage := E_ConfigStorage.AS_DINT,
        pTarget := ADR(CalendarV3.Rows[n].ActiveDays), Minimum := 0.0, Maximum := 127.0,
        RequiresReady := FALSE) AND ok;
    M_SetConfigAccess(WriteKey := key, ClassId := '', MinReadLevel := E_AccessLevel.NONE,
        MinWriteLevel := E_AccessLevel.ENGINEER);
    key := CONCAT('line.shift.', CONCAT(TO_STRING(n), '.productionTarget'));
    item := CONCAT('CalendarV3/Rows[', CONCAT(TO_STRING(n), ']/ProductionTarget'));
    label := CONCAT('std.config.shift.', CONCAT(TO_STRING(n), '.productionTarget'));
    ok := M_RegisterConfigNumber(Key := key, Item := item, LabelKey := label,
        Unit := E_EngUnit.PIECE, Kind := E_ConfigKind.LINE_CFG, Storage := E_ConfigStorage.AS_DINT,
        pTarget := ADR(CalendarV3.Rows[n].ProductionTarget), Minimum := 0.0, Maximum := 2147483647.0,
        RequiresReady := FALSE) AND ok;
    M_SetConfigAccess(WriteKey := key, ClassId := '', MinReadLevel := E_AccessLevel.NONE,
        MinWriteLevel := E_AccessLevel.ENGINEER);
END_FOR
_M_RegisterCalendar := ok;
END_METHOD

METHOD M_ShiftInterval : BOOL
VAR_INPUT
    Now : DT;
END_VAR
VAR_OUTPUT
    ShiftIndex : INT;
    StartAt : DT;
    EndAt : DT;
    Target : UDINT;
END_VAR
M_ShiftInterval := _schedule.M_Interval(Now := Now, Calendar := CalendarV3,
    ShiftIndex => ShiftIndex, StartAt => StartAt, EndAt => EndAt, Target => Target);
END_METHOD

METHOD M_StageConfigWrite : BOOL
VAR_INPUT
    Scope : STRING(255);
    WriteKey : STRING(160);
    Revision : UDINT;
    TextValue : STRING(255);
    RootReady : BOOL;
END_VAR
VAR
    i : INT;
    original : PVOID;
END_VAR
M_StageConfigWrite := FALSE;
IF NOT _batch THEN _candidate := CalendarV3; END_IF
IF NOT SUPER^.M_StageConfigWrite(Scope := Scope, WriteKey := WriteKey, Revision := Revision,
        TextValue := TextValue, RootReady := RootReady) THEN RETURN; END_IF
FOR i := 1 TO _nConfigWrite DO
    IF _pConfigWrite[i - 1].Key = WriteKey THEN
        original := _pConfigWrite[i - 1].pTarget;
        IF (original < ADR(CalendarV3)) OR (original >= ADR(CalendarV3) + SIZEOF(CalendarV3)) THEN RETURN; END_IF
        _pConfigWrite[i - 1].pTarget := ADR(_candidate) + (original - ADR(CalendarV3));
        M_StageConfigWrite := _M_StoreConfigValue(Idx := i, TextValue := TextValue, Commit := TRUE);
        _pConfigWrite[i - 1].pTarget := original;
        EXIT;
    END_IF
END_FOR
IF M_StageConfigWrite AND NOT _batch THEN
    M_StageConfigWrite := _schedule.M_Validate(Calendar := _candidate);
END_IF
END_METHOD

METHOD M_ApplyConfigWrite : BOOL
VAR_INPUT
    Scope : STRING(255);
    WriteKey : STRING(160);
    Revision : UDINT;
    TextValue : STRING(255);
    RootReady : BOOL;
END_VAR
M_ApplyConfigWrite := M_StageConfigWrite(Scope := Scope, WriteKey := WriteKey,
    Revision := Revision, TextValue := TextValue, RootReady := RootReady);
IF NOT M_ApplyConfigWrite THEN RETURN; END_IF
IF NOT _batch THEN
    CalendarV3 := _candidate;
    IF _role = E_LineRole.OWNER THEN _revision := _revision + 1; END_IF
END_IF
END_METHOD

METHOD M_BeginConfigBatch : BOOL
M_BeginConfigBatch := NOT _batch;
IF M_BeginConfigBatch THEN _candidate := CalendarV3; _batch := TRUE; END_IF
END_METHOD

METHOD M_ValidateConfigBatch : BOOL
M_ValidateConfigBatch := _batch AND _schedule.M_Validate(Calendar := _candidate);
END_METHOD

METHOD M_EndConfigBatch
_batch := FALSE;
END_METHOD

METHOD M_CommitConfigBatch : BOOL
M_CommitConfigBatch := M_ValidateConfigBatch();
IF M_CommitConfigBatch THEN
    CalendarV3 := _candidate;
    IF _role = E_LineRole.OWNER THEN _revision := _revision + 1; END_IF
END_IF
_batch := FALSE;
END_METHOD

END_FUNCTION_BLOCK

// ---- BaseClasses/FB_AsciiDeviceCM.TcPOU
// Core §3.15.1a — CM base for ASCII request/response devices over I_ByteChannel
// (vision sensors, code readers, gauges). One-outstanding-request state machine:
// SendRequest -> await terminated response -> _M_OnResponse hook; silence -> fault
// 10402. The framing and request rules are FB_AsciiLink's, shared with connectors
// (§1.1 O9); this CM adds what a CM owns: its faults and its bounded reconnect.
// Written ONCE against the neutral seam: porting = swap the channel (O4/O8).
FUNCTION_BLOCK ABSTRACT FB_AsciiDeviceCM EXTENDS FB_ControlModuleBase
VAR
    Host        : STRING(80);          // §3.8 config (per deployment)
    Port        : UINT;
    Terminator  : STRING(2) := '$R';   // CR default; device profile may override
    RespTimeout : TIME := T#2S;
    LinkState   : E_ByteChannelState;  // published (Annex D link facet)
    LastResponse: STRING(255);         // published (diagnosis)
END_VAR
VAR
    {attribute 'OPC.UA.DA' := '0'}
    _link      : FB_AsciiLink;
    _tRetry    : TON;
    _retryMs   : TIME := T#500MS;       // bounded backoff (doubles to 10s)
    _openTried : BOOL;                  // backoff spaces RE-tries; the first Open is immediate
END_VAR

;  // driven via Cyclic (base) -> OnCyclic below

// wire the transport + endpoint. Call from the profile's Setup after _M_SetName.
METHOD SetupDevice : BOOL
VAR_INPUT
    Chan : I_ByteChannel;
    DevHost : STRING(80);
    DevPort : UINT;
END_VAR
IF Chan = 0 OR DevHost = '' THEN
    _M_FaultN(PL_TcpDevReasons.DEV_CFG_INVALID, 'std.error.deviceConnectionNotConfigured');
    SetupDevice := FALSE;
    RETURN;
END_IF
_link.M_Bind(Chan := Chan);
Host := DevHost;
Port := DevPort;
SetupDevice := TRUE;
END_METHOD

// channel management + RX framing. Profiles override _M_OnResponse, not this.
METHOD PROTECTED OnCyclic : DINT
VAR
    evt : E_AsciiLinkEvent;
END_VAR
OnCyclic := SUPER^.OnCyclic();
_link.Terminator := Terminator;
_link.RespTimeout := RespTimeout;
evt := _link.M_Tick();
LinkState := _link.State;
IF LinkState = E_ByteChannelState.CLOSED THEN
    IF NOT _openTried THEN
        _openTried := TRUE;                        // first sight of CLOSED: connect NOW
        _link.M_Open(Host := Host, Port := Port);
        LinkState := _link.State;                  // a synchronous transport is OPEN this scan
    ELSE
        _tRetry(IN := TRUE, PT := _retryMs);       // failed before: bounded backoff (§3.15.2 spirit)
        IF _tRetry.Q THEN
            _tRetry(IN := FALSE);
            _link.M_Open(Host := Host, Port := Port);
            LinkState := _link.State;
            IF _retryMs < T#10S THEN
                _retryMs := _retryMs * 2;
            END_IF
        END_IF
    END_IF
ELSIF LinkState = E_ByteChannelState.OPEN THEN
    _openTried := FALSE;
    _retryMs := T#500MS;
END_IF
CASE evt OF
    E_AsciiLinkEvent.NONE:
        ;
    E_AsciiLinkEvent.RESPONSE:
        LastResponse := _link.LastResponse;
        _M_OnResponse(Response := _link.Response);
    E_AsciiLinkEvent.OVERFLOW:
        _M_FaultN(PL_TcpDevReasons.DEV_RX_OVERFLOW, 'std.error.deviceResponseOverflow');
    E_AsciiLinkEvent.CHANNEL_FAULT:
        _M_FaultN(PL_TcpDevReasons.DEV_CHANNEL_FAULT, 'std.error.transportChannelFault');
    E_AsciiLinkEvent.TIMEOUT:
        _M_FaultN(PL_TcpDevReasons.DEV_RESP_TIMEOUT, 'std.error.deviceResponseTimeout');
ELSE
    _M_FaultN(PL_TcpDevReasons.DEV_CHANNEL_FAULT, 'std.error.byteChannelStateInvalid');
END_CASE
END_METHOD

// issue one request (terminator appended). FALSE if not connected or one pending.
METHOD SendRequest : BOOL
VAR_INPUT
    Text : STRING(250);
END_VAR
IF NOT _link.M_IsOpen() THEN
    _M_FaultN(PL_TcpDevReasons.DEV_NOT_CONNECTED, 'std.error.deviceNotConnected');
    SendRequest := FALSE;
    RETURN;
END_IF
// A pending request is the one-outstanding contract, not a fault: refused quietly.
_link.Terminator := Terminator;
SendRequest := _link.M_Send(Text := Text);
END_METHOD

// profile hook: parse one terminated response. Raise DEV_PROTOCOL on garbage.
METHOD PROTECTED _M_OnResponse
VAR_INPUT
    Response : STRING(255);
END_VAR
;
END_METHOD

END_FUNCTION_BLOCK

// ---- Connectivity/FB_AsciiLink.TcPOU
// Core §3.15.1a - ASCII request/response over I_ByteChannel, written ONCE: terminator
// framing, the one-outstanding-request rule, the receive bound and the response
// timeout. It owns no open policy and raises nothing: each tick returns an event,
// and its owner decides what that means - FB_AsciiDeviceCM faults and reconnects
// on its own backoff; a connector on FB_DeviceConnectorBase leaves session,
// heartbeat and reconnect to that base (§3.15.2). One framing, two owners (§1.1 O9).
FUNCTION_BLOCK FB_AsciiLink
VAR_INPUT
    Terminator  : STRING(2) := '$R';   // CR default; a device profile may override
    RespTimeout : TIME := T#2S;
END_VAR
VAR_OUTPUT
    State        : E_ByteChannelState; // last observed transport state
    Pending      : BOOL;               // one request outstanding
    Response     : STRING(255);        // the response of the last RESPONSE event
    LastResponse : STRING(255);        // kept until the next response (diagnosis)
END_VAR
VAR
    {attribute 'OPC.UA.DA' := '0'}
    _chan  : I_ByteChannel;
    _rx    : STRING(255);
    _tResp : TON;
END_VAR

;  // driven through M_Tick by its owner

METHOD M_Bind : BOOL
VAR_INPUT
    Chan : I_ByteChannel;
END_VAR
_chan := Chan;
M_Bind := (Chan <> 0);
END_METHOD

// TRUE when the transport accepted the open (OPENING, or OPEN at once on a
// synchronous transport). Whether it then comes up is observed over scans.
METHOD M_Open : BOOL
VAR_INPUT
    Host : STRING(80);
    Port : UINT;
END_VAR
M_Open := FALSE;
IF _chan = 0 THEN
    RETURN;
END_IF
_chan.Open(Host := Host, Port := Port);
State := _chan.State();
M_Open := (State = E_ByteChannelState.OPEN) OR (State = E_ByteChannelState.OPENING);
END_METHOD

METHOD M_Close : BOOL
M_Close := FALSE;
Pending := FALSE;
_tResp(IN := FALSE);
_rx := '';
IF _chan = 0 THEN
    RETURN;
END_IF
M_Close := _chan.Close();
State := _chan.State();
END_METHOD

// LIVE transport state (the published State is one scan old).
METHOD M_IsOpen : BOOL
M_IsOpen := FALSE;
IF _chan = 0 THEN
    RETURN;
END_IF
M_IsOpen := (_chan.State() = E_ByteChannelState.OPEN);
END_METHOD

// Issue one request (terminator appended). FALSE when there is no channel, it is
// not OPEN, or a request is already outstanding - refused, never queued.
METHOD M_Send : BOOL
VAR_INPUT
    Text : STRING(250);
END_VAR
M_Send := FALSE;
// The null test is its own statement: TwinCAT does not short-circuit by default,
// so folding it into the next condition would still call State() on a null
// interface and fault the runtime.
IF _chan = 0 THEN
    RETURN;
END_IF
// LIVE state: the cached State is one scan old and would reject a request issued
// in the same scan the transport opened.
IF _chan.State() <> E_ByteChannelState.OPEN THEN
    RETURN;
END_IF
IF Pending THEN
    RETURN;
END_IF
Pending := _chan.Send(Text := CONCAT(Text, Terminator));
M_Send := Pending;
END_METHOD

// Run the transport one scan: drain, frame one response, watch the timeout.
METHOD M_Tick : E_AsciiLinkEvent
VAR
    pos : INT;
END_VAR
M_Tick := E_AsciiLinkEvent.NONE;
IF _chan = 0 THEN
    RETURN;
END_IF
_chan.Tick();
State := _chan.State();
CASE State OF
    E_ByteChannelState.CLOSED, E_ByteChannelState.OPENING:
        ;                                       // the owner decides when to open
    E_ByteChannelState.OPEN:
        _chan.Poll(Buffer := _rx);
        pos := FIND(_rx, Terminator);
        IF pos > 0 THEN
            Response := LEFT(_rx, pos - 1);
            _rx := DELETE(_rx, pos + LEN(Terminator) - 1, 1);
            Pending := FALSE;
            _tResp(IN := FALSE);
            LastResponse := Response;
            M_Tick := E_AsciiLinkEvent.RESPONSE;
            RETURN;
        ELSIF LEN(_rx) >= 250 THEN
            _rx := '';
            M_Tick := E_AsciiLinkEvent.OVERFLOW;
            RETURN;                             // first-out; the timeout still runs next scan
        END_IF
    E_ByteChannelState.FAULT:
        Pending := FALSE;
        _tResp(IN := FALSE);
        _chan.Close();
        M_Tick := E_AsciiLinkEvent.CHANNEL_FAULT;
        RETURN;
ELSE
    _chan.Close();
    M_Tick := E_AsciiLinkEvent.INVALID_STATE;
    RETURN;
END_CASE
_tResp(IN := Pending, PT := RespTimeout);
IF _tResp.Q THEN
    Pending := FALSE;
    _tResp(IN := FALSE);
    M_Tick := E_AsciiLinkEvent.TIMEOUT;
END_IF
END_METHOD

END_FUNCTION_BLOCK

// ---- Connectivity/F_AppendTopologyConfig.TcPOU
// Core §3.10.2/§10.5.1 — export the activation-static fieldbus identity (tags,
// addresses, wiring, hierarchy) into the config manifest. The live members
// (State/LinkOk/values/force/quality/fault) stay cyclically published; the
// static members carry OPC.UA.DA=0 in ST_BusNode/ST_IoChannel and reach the
// HMI only through this walk. Item fragments use the server's array naming
// (Nodes/Nodes[i]/..., Channels/Channels[j]/...) under the reserved scope
// '#Fieldbus' so a generic client can rebuild the exact browse paths.
// Only populated slots are exported — the empty tail of the bounded table
// costs nothing on the wire.
FUNCTION F_AppendTopologyConfig : BOOL
VAR_IN_OUT
    Topology : ST_FieldbusTopology;
    Pager    : FB_ConfigPager;
END_VAR
VAR
    i, j       : INT;
    nodeBase   : STRING(255);
    chanBase   : STRING(255);
    item       : STRING(255);
    forceableText : STRING(5);
END_VAR
VAR CONSTANT
    SCOPE_FIELDBUS : STRING(16) := '#Fieldbus';
END_VAR

F_AppendTopologyConfig := TRUE;
FOR i := 1 TO Topology.NodeCount DO
    IF (i < 1) OR (i > PL_Fraktal.MAX_BUS_NODES) THEN
        EXIT;                                       // defensive bound (§5.6)
    END_IF
    nodeBase := CONCAT('Nodes/Nodes[', CONCAT(TO_STRING(i), ']/'));
    Pager.M_Append(Scope := SCOPE_FIELDBUS,
        Item := CONCAT(nodeBase, 'Name'), ValueText := Topology.Nodes[i].Name);
    Pager.M_Append(Scope := SCOPE_FIELDBUS,
        Item := CONCAT(nodeBase, 'DescriptionKey'),
        ValueText := Topology.Nodes[i].DescriptionKey);
    Pager.M_Append(Scope := SCOPE_FIELDBUS,
        Item := CONCAT(nodeBase, 'TypeId'), ValueText := Topology.Nodes[i].TypeId);
    Pager.M_Append(Scope := SCOPE_FIELDBUS,
        Item := CONCAT(nodeBase, 'Address'), ValueText := Topology.Nodes[i].Address);
    Pager.M_AppendNumber(Scope := SCOPE_FIELDBUS,
        Item := CONCAT(nodeBase, 'ParentIdx'),
        Number := TO_DINT(Topology.Nodes[i].ParentIdx));
    Pager.M_AppendNumber(Scope := SCOPE_FIELDBUS,
        Item := CONCAT(nodeBase, 'ChannelCount'),
        Number := TO_DINT(Topology.Nodes[i].ChannelCount));
    FOR j := 1 TO Topology.Nodes[i].ChannelCount DO
        IF (j < 1) OR (j > PL_Fraktal.MAX_NODE_CHANNELS) THEN
            EXIT;                                   // defensive bound (§5.6)
        END_IF
        chanBase := CONCAT(nodeBase,
            CONCAT('Channels/Channels[', CONCAT(TO_STRING(j), ']/')));
        Pager.M_Append(Scope := SCOPE_FIELDBUS,
            Item := CONCAT(chanBase, 'Name'),
            ValueText := Topology.Nodes[i].Channels[j].Name);
        Pager.M_Append(Scope := SCOPE_FIELDBUS,
            Item := CONCAT(chanBase, 'DescriptionKey'),
            ValueText := Topology.Nodes[i].Channels[j].DescriptionKey);
        Pager.M_Append(Scope := SCOPE_FIELDBUS,
            Item := CONCAT(chanBase, 'Address'),
            ValueText := Topology.Nodes[i].Channels[j].Address);
        Pager.M_Append(Scope := SCOPE_FIELDBUS,
            Item := CONCAT(chanBase, 'Path'),
            ValueText := Topology.Nodes[i].Channels[j].Path);
        Pager.M_Append(Scope := SCOPE_FIELDBUS,
            Item := CONCAT(chanBase, 'ModulePath'),
            ValueText := Topology.Nodes[i].Channels[j].ModulePath);
        Pager.M_AppendNumber(Scope := SCOPE_FIELDBUS,
            Item := CONCAT(chanBase, 'Dir'),
            Number := TO_DINT(Topology.Nodes[i].Channels[j].Dir));
        Pager.M_AppendNumber(Scope := SCOPE_FIELDBUS,
            Item := CONCAT(chanBase, 'Kind'),
            Number := TO_DINT(Topology.Nodes[i].Channels[j].Kind));
        Pager.M_Append(Scope := SCOPE_FIELDBUS,
            Item := CONCAT(chanBase, 'Unit'),
            ValueText := Topology.Nodes[i].Channels[j].Unit);
        IF Topology.Nodes[i].Channels[j].Forceable THEN
            forceableText := 'TRUE';
        ELSE
            forceableText := 'FALSE';
        END_IF
        Pager.M_Append(Scope := SCOPE_FIELDBUS,
            Item := CONCAT(chanBase, 'Forceable'), ValueText := forceableText);
    END_FOR
END_FOR

END_FUNCTION

// ---- Connectivity/FB_DeviceConnectorBase.TcPOU
// Core §3.15 written once: session + heartbeat + LinkTimeout loss confirm +
// bounded exponential backoff reconnect + NO self-resume of dependents (that is
// the fronting CM's contract). A transport implements only _M_Open/_M_Close/
// _M_HbStart/_M_HbPoll. Row T7 of §5.7 is proven here once.
FUNCTION_BLOCK ABSTRACT FB_DeviceConnectorBase IMPLEMENTS I_DeviceConnector
VAR_INPUT
    HbPeriod    : TIME := T#1S;
    LinkTimeout : TIME := T#3S;
    BackoffMin  : TIME := T#500MS;
    BackoffMax  : TIME := T#10S;
    Reaction    : E_LinkReaction := E_LinkReaction.HOLD;   // consumed by the fronting CM
END_VAR
VAR
    _name      : STRING(80);
    _sessionUp : BOOL;
    _linked    : BOOL;
    _hbBusy    : BOOL;
    _lastSeen  : DT;
    _diag      : ST_Diagnostic;
    _tHb, _tLoss, _tBk : TON;
    _backoffMs : DINT;
END_VAR

Cyclic();

METHOD Connect : BOOL
Connect := _M_TryOpen();
END_METHOD

METHOD Cyclic : BOOL
IF NOT _sessionUp THEN
    // bounded exponential backoff (§3.15) — never a tight reconnect loop
    _tBk(IN := TRUE, PT := DINT_TO_TIME(_backoffMs));
    IF _tBk.Q THEN
        _tBk(IN := FALSE);
        IF NOT _M_TryOpen() THEN
            _backoffMs := MIN(_backoffMs * 2, TIME_TO_DINT(BackoffMax));
        END_IF
    END_IF
    Cyclic := TRUE;
    RETURN;
END_IF
// heartbeat: issue when due, poll while busy
IF NOT _hbBusy THEN
    _tHb(IN := TRUE, PT := HbPeriod);
    IF _tHb.Q THEN
        _tHb(IN := FALSE);
        _hbBusy := _M_HbStart();
    END_IF
ELSE
    CASE _M_HbPoll() OF
        E_HbResult.OK:
            _hbBusy := FALSE;
            _linked := TRUE;
            _lastSeen := F_Now();                 // §2.7
            _diag.ReasonCode := E_Reason.NONE;
            _diag.Description := '';
            _tLoss(IN := FALSE);                  // healthy beat resets loss confirm
        E_HbResult.FAIL:
            _hbBusy := FALSE;
            _M_Lost(E_Reason.DEVICE_PROTOCOL_ERROR, 'std.error.heartbeatBadReply');
            Cyclic := TRUE;
            RETURN;
        E_HbResult.PENDING:
            ;                                      // request still in flight
    ELSE
        _hbBusy := FALSE;
        _M_Lost(E_Reason.DEVICE_PROTOCOL_ERROR, 'std.error.heartbeatResultInvalid');
        Cyclic := TRUE;
        RETURN;
    END_CASE
END_IF
// confirm loss only after LinkTimeout without a healthy beat (§3.15.2)
_tLoss(IN := TRUE, PT := LinkTimeout);
IF _tLoss.Q THEN
    _M_Lost(E_Reason.LINK_TIMEOUT, 'std.error.heartbeatLapsed');
END_IF
Cyclic := TRUE;
END_METHOD

METHOD Disconnect : BOOL
_M_Close();
_sessionUp := FALSE;
_linked := FALSE;
Disconnect := TRUE;
END_METHOD

// I_Module command-release seam. The connector owns no PLCopen Execute latch;
// the fronting Control Module owns and releases the dependent device command.
// Disconnecting here would defeat the mandatory bounded reconnect policy (Core §3.15.2).
METHOD M_ReleaseCommand : BOOL
M_ReleaseCommand := TRUE;
END_METHOD

METHOD GetFaultSummary : ST_Diagnostic
GetFaultSummary := _diag;
END_METHOD

METHOD PrepareRecipe : BOOL
VAR_INPUT
    Model : ST_ModelId;
END_VAR
PrepareRecipe := TRUE;
END_METHOD

METHOD CommitRecipe
END_METHOD

METHOD AbortRecipe
END_METHOD

METHOD Setup : BOOL
VAR_INPUT
    Name : STRING(80);
END_VAR
_name := Name;
_backoffMs := TIME_TO_DINT(BackoffMin);
Setup := TRUE;
END_METHOD

METHOD PROTECTED ABSTRACT _M_Close : BOOL
END_METHOD

// PENDING while in flight; OK resets loss confirm; FAIL = protocol error
METHOD PROTECTED ABSTRACT _M_HbPoll : E_HbResult
END_METHOD

METHOD PROTECTED ABSTRACT _M_HbStart : BOOL
END_METHOD

// stamp the link first-out, drop the session; reconnection is backoff-bounded,
// resumption of dependent commands is NEVER automatic (§3.15/§9.3)
METHOD PROTECTED _M_Lost
VAR_INPUT
    Reason : E_Reason;
    Text   : STRING(255);
END_VAR
IF _diag.ReasonCode <> Reason THEN
    _diag.Since := F_Now();
    _diag.TimeSynchronized := F_TimeSynchronized();
END_IF
_diag.ReasonCode  := Reason;
_diag.Description := Text;
_diag.SourcePath  := _name;
_diag.Severity    := E_Severity.MED;
_diag.Category    := E_Category.SYSTEM;
F_RationalizeDiagnostic(Diag := _diag);
_linked := FALSE;
_hbBusy := FALSE;
_M_Close();
_sessionUp := FALSE;
END_METHOD

METHOD PROTECTED ABSTRACT _M_Open : BOOL
END_METHOD

METHOD PROTECTED _M_TryOpen : BOOL
IF _M_Open() THEN
    _sessionUp := TRUE;
    _backoffMs := TIME_TO_DINT(BackoffMin);
    _M_TryOpen := TRUE;
ELSE
    _M_TryOpen := FALSE;
END_IF
END_METHOD

PROPERTY FaultActive : BOOL
GET
FaultActive := (NOT _linked) AND (_diag.ReasonCode <> E_Reason.NONE);
END_GET
END_PROPERTY

// The connector reports link state/faults. HOLD is a configured loss reaction
// interpreted by the fronting Control Module; it is not connector lifecycle state.
PROPERTY HoldActive : BOOL
GET
HoldActive := FALSE;
END_GET
END_PROPERTY

PROPERTY LastSeen : DT
GET
LastSeen := _lastSeen;
END_GET
END_PROPERTY

PROPERTY Linked : BOOL
GET
Linked := _linked;
END_GET
END_PROPERTY

PROPERTY LinkReason : ST_Diagnostic
GET
LinkReason := _diag;
END_GET
END_PROPERTY

PROPERTY ModuleType : E_ModuleType
GET
ModuleType := E_ModuleType.CONTROL_MODULE;
END_GET
END_PROPERTY

PROPERTY Name : STRING(80)
GET
Name := _name;
END_GET
END_PROPERTY

PROPERTY State : E_ExecState
GET
State := SEL(FaultActive, E_ExecState.READY, E_ExecState.ERROR);
END_GET
END_PROPERTY

END_FUNCTION_BLOCK

// ---- Connectivity/FB_EcBusHealth.TcPOU
// Core §10.5.1 infrastructure service: read the REAL, live state of every
// EtherCAT slave directly from the fieldbus master (Tc2_EtherCAT) and publish it
// per node, so the HMI fieldbus tree mirrors XAE — independent of any Control-On
// or safety verdict. Auto-detects from hardware: the project supplies only the
// master AmsNetId ('' = local CPU) and how its topology node indices line up
// with the master's slave ordering (one offset), not per-node wiring.
//
// This is not a module tier and owns no process image. It calls
// FB_IoTopologyPublisher.M_SetNodeState for each mapped node.
FUNCTION_BLOCK FB_EcBusHealth
VAR
    {attribute 'OPC.UA.DA' := '0'}
    _pub : POINTER TO FB_IoTopologyPublisher;
    _netId : T_AmsNetId;          // EtherCAT MASTER device AmsNetId (see Setup)
    _firstSlaveNode : INT;        // topology node index of master slave #1
    _slaveCount : INT;            // how many slaves the master is asked about
    _masterNode : INT;            // topology node index of the master itself (0 = none)
    _attached : BOOL;

    // §10.5.1 — which topology node each MASTER SLAVE INDEX belongs to.
    // _slaveNode[i] = topology node of the master's slave i (0 = unmapped).
    //
    // The master enumerates only devices with an EtherCAT slave controller on
    // the process-data ring. A bus coupler (EK1200) and a passive end cap
    // (EL9011) are in the project tree and in the catalog, but the master never
    // lists them -- so "catalog position" and "master slave index" are NOT the
    // same sequence. Assuming they were shifted every state by one: the press
    // bench published the EL1809's state onto the coupler, the EL2809's onto the
    // EL1809, the EL6001's onto the EL2809, and left the real EL6001 and the end
    // cap reading OFFLINE while all three cards were in OP. A wrong state on the
    // right node is worse than no state: it is a plausible lie.
    //
    // Setup's FirstSlaveNode/SlaveCount form still works and fills this map
    // consecutively -- correct whenever every catalogued node really is a slave.
    _slaveNode : ARRAY[1..PL_Fraktal.MAX_BUS_NODES] OF INT;
    // Topology nodes that are catalogued but are NOT on the master's slave list
    // (couplers, end caps). Their state is inferred, never invented: they carry
    // the bus and are reachable exactly when the slaves behind them answer.
    _passiveNode : ARRAY[1..PL_Fraktal.MAX_BUS_NODES] OF INT;
    _passiveCount : INT;

    // Auto-detection of the EtherCAT master's AmsNetId (no project wiring): the
    // master's NetId is the local AMS NetId with the last two bytes replaced by
    // 2.1 (Beckhoff convention -- a PC 'a.b.c.d.1.1' has its EtherCAT master at
    // 'a.b.c.d.2.1'; the InfoSys FB_EcGetAllSlaveStates example uses exactly this
    // pairing). Overridable via Setup for non-standard configurations.
    {attribute 'OPC.UA.DA' := '0'}
    _fbLocalNetId : Tc2_Utilities.FB_GetLocalAmsNetId;
    _autoDetect : BOOL;           // TRUE = derive the master NetId at runtime
    {attribute 'OPC.UA.DA' := '0'}
    _netIdArr : T_AmsNetIdArr;    // scratch for the derived master NetId

    {attribute 'OPC.UA.DA' := '0'}
    _fbStates : Tc2_EtherCAT.FB_EcGetAllSlaveStates;
    // Bounded state buffer, one ST_EcSlaveState (deviceState + linkState) per
    // slave. Beckhoff declares pStateBuf as ARRAY[0..EC_MAX_SLAVES], so this
    // buffer is ZERO-BASED: slave i (1..n, master scan order) is _stateBuf[i-1].
    {attribute 'OPC.UA.DA' := '0'}
    _stateBuf : ARRAY[0..PL_Fraktal.MAX_BUS_NODES] OF Tc2_EtherCAT.ST_EcSlaveState;
    _step : INT;
    _tPoll : TON;
    // Demand gating (§10.5.1 diagnostic surface): only scan while a consumer
    // asks. _firstScanDone lets one scan run after Setup so M_BusOk() — which
    // feeds control logic, not a view — is never based on unread hardware.
    _scanRequested : BOOL;
    _firstScanDone : BOOL;

    // §8.12/§10.5 master health. Unlike the per-slave picture it is NOT
    // demand-gated: alarms and M_BusOk consume it every scan, so it is sampled
    // once a second whether or not anyone has the bus view open.
    {attribute 'OPC.UA.DA' := '0'}
    _fbDevState : Tc2_EtherCAT.FB_EcGetMasterDevState;
    {attribute 'OPC.UA.DA' := '0'}
    _fbFrames : Tc2_EtherCAT.FB_EcMasterFrameStatistic;
    {attribute 'OPC.UA.DA' := '0'}
    _fbCrc : Tc2_EtherCAT.FB_EcGetAllSlaveCrcErrors;
    {attribute 'OPC.UA.DA' := '0'}
    _crcBuf : ARRAY[0..PL_Fraktal.MAX_BUS_NODES] OF DWORD;
    _mPhase : INT;
    _mPoll : TON;
    _mSampled : BOOL;
    _mSampledAt : TIME;
    _mBaselined : BOOL;
    _mWindowStart : TIME;
    _mLostBase : UDINT;
    _mCrcBase : UDINT;
    _mLastWindowLost : UDINT;
    _mLastWindowCrc : UDINT;
END_VAR
VAR CONSTANT
    // Tc2_EtherCAT master device-state bits (F_ConvMasterDevStateToString): link
    // error 0x0001, I/O locked 0x0002, out of send resources 0x0010, watchdog
    // 0x0020, driver missing 0x0040, I/O reset 0x0080, a device in INIT/PRE-OP/
    // SAFE-OP 0x0100/0x0200/0x0400, a device in error 0x0800. The redundancy-only
    // bits 0x0004/0x0008 are not faults of a working line; DC is reported apart.
    MASTER_FAULT_BITS : WORD := 16#0FF3;
    MASTER_DC_NOT_IN_SYNC : WORD := 16#1000;
    MASTER_POLL : TIME := T#1S;
    MASTER_WINDOW : TIME := T#10S;
    MASTER_FRESH_FOR : TIME := T#3S;
END_VAR
VAR_OUTPUT
    // Diagnostics so a fieldbus read failure is visible instead of silently
    // showing every node as faulted. Published for the HMI/engineer.
    ReadOk : BOOL;                // last slave-state read succeeded
    LastErrorId : UDINT;          // ADS error of the last failed read (0 = none)
    SlavesReported : UINT;        // slaves the master reports (nSlaves output)
    NetIdMissing : BOOL;          // TRUE = InfoData.AmsNetId not linked (all zero)
    MasterNetId : T_AmsNetId;     // the resolved master NetId actually being used
    // TRUE = the master reports a different slave count than the project
    // topology declares (missing/extra hardware, or a config not activated).
    // §10.5.1: an unmatched mapping is a commissioning error, never guessed.
    CountMismatch : BOOL;

    // ---- Raw read-back diagnostics (commissioning aid) --------------------
    // The decoded E_NodeState alone cannot distinguish "the master said INIT"
    // from "we indexed or decoded it wrong". These publish the EXACT bytes the
    // master returned plus how each was interpreted, so a disagreement with XAE
    // is attributable to hardware, indexing, or decode without attaching a
    // debugger. Deliberately PUBLISHED (no 'OPC.UA.DA' := '0'): the point is
    // that an engineer can read them remotely over ADS/OPC UA.
    // Read them as: slot k holds slave k (master scan order), which this
    // library maps to topology node DiagNodeIndex[k].
    DiagRawDeviceState : ARRAY[1..8] OF BYTE;   // deviceState byte, as received
    DiagRawLinkState : ARRAY[1..8] OF BYTE;     // linkState byte, as received
    DiagDecodedState : ARRAY[1..8] OF INT;      // E_NodeState after decoding
    DiagNodeIndex : ARRAY[1..8] OF INT;         // topology node each slave maps to
    DiagBufferBytes : UDINT;                    // cbBufLen passed to the FB
    DiagEntrySize : UDINT;                      // SIZEOF(ST_EcSlaveState)
    DiagScanCount : UDINT;                      // completed reads (proves polling)
    DiagScanRequested : BOOL;                   // the §10.5.1 demand-gate state
    DiagFirstScanDone : BOOL;

    // ---- Master health (§8.12/§10.5): sampled every second, never gated ----
    MasterAvailable : BOOL;     // state, frame and CRC counters read within 3 s
    MasterDevState  : WORD;     // raw master device state (F_ConvMasterDevStateToString)
    MasterHealthy   : BOOL;     // available and no MASTER_FAULT_BITS set
    LostFrameCount  : UDINT;    // lost cyclic+queued frames: current or last 10 s window
    SlaveErrorCount : UDINT;    // summed slave CRC errors: current or last 10 s window
    DcSynchronized  : BOOL;     // available and DC not reported out of sync
    MasterErrorId   : UDINT;    // ADS error of the last failed master read (0 = none)
END_VAR

;

// Bind the publisher and describe how topology nodes map to master slaves.
// MasterNetIdArr = OPTIONAL override for the EtherCAT master's AmsNetId. Pass all
//   zeros (the normal case, e.g. an unassigned T_AmsNetIdArr) to AUTO-DETECT it at
//   runtime: the library reads the local AMS NetId and applies the Beckhoff master
//   convention (last two bytes -> 2.1), so no project wiring, no XAE checkbox and
//   no hand-typed address are needed. Supply a value only for a non-standard
//   configuration (e.g. a remote master, or several masters on one PC), typically
//   by linking that master's InfoData.AmsNetId.
// FirstSlaveNode = topology index of the first EtherCAT slave (the coupler);
// SlaveCount = number of consecutive topology nodes that are real slaves, in
// master scan order; MasterNodeIndex = topology index of the EtherCAT master
// itself, or 0 if not represented.
METHOD Setup : BOOL
VAR_INPUT
    Publisher : REFERENCE TO FB_IoTopologyPublisher;
    MasterNetIdArr : T_AmsNetIdArr;
    FirstSlaveNode : INT;
    SlaveCount : INT;
    MasterNodeIndex : INT;
END_VAR
VAR
    i : INT;
    anyNonZero : BOOL;
END_VAR
// All-zero (or omitted) = auto-detect; any explicit value is used verbatim.
anyNonZero := FALSE;
FOR i := 0 TO 5 DO
    IF MasterNetIdArr[i] <> 0 THEN
        anyNonZero := TRUE;
    END_IF
END_FOR

_attached := __ISVALIDREF(Publisher)
    AND (FirstSlaveNode >= 1)
    AND (SlaveCount >= 0)
    AND (SlaveCount <= PL_Fraktal.MAX_BUS_NODES);
IF _attached THEN
    _pub := ADR(Publisher);
    _autoDetect := NOT anyNonZero;
    IF anyNonZero THEN
        // Tc2_System helper: byte array -> 'a.b.c.d.e.f' string.
        _netId := Tc2_System.F_CreateAmsNetId(nIds := MasterNetIdArr);
        MasterNetId := _netId;
        NetIdMissing := FALSE;
        _step := 0;
    ELSE
        // Resolve the local NetId first (step -10), then start polling.
        _netId := '';
        MasterNetId := '';
        NetIdMissing := TRUE;   // cleared once auto-detection succeeds
        _step := -10;
    END_IF
    _firstSlaveNode := FirstSlaveNode;
    _slaveCount := SlaveCount;
    _masterNode := MasterNodeIndex;
    // Consecutive default: master slave i -> topology node FirstSlaveNode+i-1.
    // Correct only when EVERY catalogued node in that window is a real slave;
    // call M_MapSlaveNode to state the mapping explicitly when it is not.
    _passiveCount := 0;
    FOR i := 1 TO PL_Fraktal.MAX_BUS_NODES DO
        IF i <= _slaveCount THEN
            _slaveNode[i] := _firstSlaveNode + i - 1;
        ELSE
            _slaveNode[i] := 0;
        END_IF
        _passiveNode[i] := 0;
    END_FOR
END_IF
Setup := _attached;
END_METHOD

// §10.5.1 — state explicitly which topology node the master's slave [SlaveIndex]
// is, for a bus whose catalog is NOT one-to-one with the master's slave list.
//
// The master enumerates only devices with an EtherCAT slave controller on the
// process-data ring. A bus coupler or a passive end cap appears in the project
// tree and in the catalog, but never in that list, so the default consecutive
// mapping shifts every state onto its neighbour. Call this once per real slave,
// after Setup, and the shift is impossible:
//
//   _busHealth.Setup(..., FirstSlaveNode := 2, SlaveCount := 3, MasterNodeIndex := 1);
//   _busHealth.M_MapSlaveNode(SlaveIndex := 1, NodeIndex := 3);  // EL1809
//   _busHealth.M_MapSlaveNode(SlaveIndex := 2, NodeIndex := 4);  // EL2809
//   _busHealth.M_MapSlaveNode(SlaveIndex := 3, NodeIndex := 5);  // EL6001
//   _busHealth.M_MapPassiveNode(NodeIndex := 2);                 // EK1200 coupler
//   _busHealth.M_MapPassiveNode(NodeIndex := 6);                 // EL9011 end cap
METHOD M_MapSlaveNode : BOOL
VAR_INPUT
    SlaveIndex : INT;   // 1-based index in the master's slave list
    NodeIndex : INT;    // topology node this slave IS (0 clears the mapping)
END_VAR
M_MapSlaveNode := _attached
    AND (SlaveIndex >= 1) AND (SlaveIndex <= PL_Fraktal.MAX_BUS_NODES)
    AND (NodeIndex >= 0);
IF M_MapSlaveNode THEN
    _slaveNode[SlaveIndex] := NodeIndex;
END_IF
END_METHOD

// §10.5.1 — declare a catalogued node that carries the bus but is NOT a slave
// the master enumerates (bus coupler, end cap, power feed).
//
// Its state is INFERRED, never invented: the devices behind it can only answer
// if it is passing traffic, so it is OPERATIONAL exactly when the read
// succeeded and at least one real slave reported. Without this it would sit at
// OFFLINE forever on a perfectly healthy bus -- which is the same "plausible
// lie" the positional mapping produced, just in the other direction.
METHOD M_MapPassiveNode : BOOL
VAR_INPUT
    NodeIndex : INT;
END_VAR
M_MapPassiveNode := _attached
    AND (NodeIndex >= 1)
    AND (_passiveCount < PL_Fraktal.MAX_BUS_NODES);
IF M_MapPassiveNode THEN
    _passiveCount := _passiveCount + 1;
    _passiveNode[_passiveCount] := NodeIndex;
END_IF
END_METHOD

// Non-blocking cyclic refresh: (re)issue the slave-state read at a bounded rate,
// then publish each node's real state. On a read error every mapped node is
// marked OFFLINE (fail-visible: an unreachable master is not "operational").
METHOD M_Refresh
VAR
    i : INT;
    node : INT;
    mapped : E_NodeState;
    linkOk : BOOL;
    reported : INT;   // slaves the master actually returned this read
END_VAR
IF NOT _attached THEN
    RETURN;
END_IF

// Mirror the gate state every cycle so "why is it not updating?" is answerable
// from published data alone: from the outside a PARKED scanner and a STUCK one
// look identical.
DiagScanRequested := _scanRequested;
DiagFirstScanDone := _firstScanDone;

// Master health first: it is consumed by alarms and M_BusOk, never parked.
_M_SampleMaster();

// §10.5.1 is a DIAGNOSTIC surface: the bus picture is only consumed while the
// fieldbus view is open. Polling the master every 250 ms regardless costs ADS
// bandwidth and PLC time for data nobody is reading, so the read is demand-gated
// (M_RequestScan, set by the HMI opening the view / a mailbox request). While no
// consumer is active the state machine idles and the last published states are
// held — they are not falsified, just not refreshed.
// Exception: the FIRST scan after Setup always runs, so M_BusOk() (a control
// input, not a view) has real data without anyone opening the HMI.
IF NOT _scanRequested AND _firstScanDone THEN
    _tPoll(IN := FALSE);
    RETURN;
END_IF

// Drive the async read. Re-trigger on a slow poll so a stuck call cannot pin the
// task; FB_EcGetAllSlaveStates is edge-triggered by bExecute. The slave count is
// implied by cbBufLen (nSlave * SIZEOF(ST_EcSlaveState)); there is no count input.
CASE _step OF
    -10:
        // Auto-detect: ask the router for this PC's AmsNetId.
        _fbLocalNetId(bExecute := FALSE);
        _fbLocalNetId(bExecute := TRUE);
        _step := -5;
    -5:
        _fbLocalNetId(bExecute := FALSE);
        IF NOT _fbLocalNetId.bBusy THEN
            IF _fbLocalNetId.bError THEN
                // Cannot resolve: stay fail-visible and retry on the next poll.
                ReadOk := FALSE;
                LastErrorId := _fbLocalNetId.nErrId;
                NetIdMissing := TRUE;
                _M_PublishAllOffline();
                _step := -10;
            ELSE
                // Beckhoff convention: the EtherCAT master of a PC 'a.b.c.d.1.1'
                // is 'a.b.c.d.2.1'. Keep the first four bytes, force 2.1.
                _netIdArr := _fbLocalNetId.AddrBytes;
                _netIdArr[4] := 2;
                _netIdArr[5] := 1;
                _netId := Tc2_System.F_CreateAmsNetId(nIds := _netIdArr);
                MasterNetId := _netId;
                NetIdMissing := FALSE;
                _step := 0;
            END_IF
        END_IF
    0:
        _fbStates(bExecute := FALSE);
        _fbStates(sNetId := _netId,
            pStateBuf := ADR(_stateBuf),
            cbBufLen := TO_UDINT(_slaveCount) * SIZEOF(Tc2_EtherCAT.ST_EcSlaveState),
            bExecute := (_slaveCount > 0));
        _step := 10;
    10:
        _fbStates(bExecute := FALSE);
        IF NOT _fbStates.bBusy THEN
            // Publish diagnostics every cycle so a failing read is visible.
            ReadOk := NOT _fbStates.bError;
            LastErrorId := _fbStates.nErrId;
            SlavesReported := _fbStates.nSlaves;
            IF NOT _fbStates.bError THEN
                // Only the first nSlaves buffer entries were written by the
                // master; the rest keep their previous/zero content. Decoding a
                // zeroed entry yields linkState 0, which reads as "link OK" — a
                // FAIL-OPEN that showed absent slaves as healthy. Publish only
                // what the master actually reported and mark the surplus
                // OFFLINE + link down (fail-closed).
                reported := TO_INT(_fbStates.nSlaves);
                IF reported > _slaveCount THEN
                    reported := _slaveCount;
                END_IF
                CountMismatch := (TO_INT(_fbStates.nSlaves) <> _slaveCount);
                // Commissioning trace: record what the master ACTUALLY returned,
                // before any interpretation, for the first 8 slaves.
                DiagScanCount := DiagScanCount + 1;
                DiagBufferBytes := TO_UDINT(_slaveCount) * SIZEOF(Tc2_EtherCAT.ST_EcSlaveState);
                DiagEntrySize := SIZEOF(Tc2_EtherCAT.ST_EcSlaveState);
                FOR i := 1 TO 8 DO
                    IF i <= _slaveCount THEN
                        DiagRawDeviceState[i] := _stateBuf[i - 1].deviceState;
                        DiagRawLinkState[i] := _stateBuf[i - 1].linkState;
                        DiagNodeIndex[i] := _slaveNode[i];
                    ELSE
                        DiagRawDeviceState[i] := 0;
                        DiagRawLinkState[i] := 0;
                        DiagNodeIndex[i] := 0;
                    END_IF
                END_FOR
                FOR i := 1 TO _slaveCount DO
                    // The topology node this master slave IS -- from the
                    // explicit map, not from position (see _slaveNode).
                    node := _slaveNode[i];
                    IF i <= reported THEN
                        // pStateBuf is ARRAY[0..EC_MAX_SLAVES]: slave i is at i-1.
                        // Decode the deviceState byte (AL state + flags).
                        mapped := _M_MapSlaveState(DeviceState := _stateBuf[i - 1].deviceState);
                        // linkState low nibble = link condition; 0 = OK.
                        linkOk := (_stateBuf[i - 1].linkState AND 16#0F) = 0;
                    ELSE
                        // Declared in the topology but never reported by the
                        // master: it is not on the bus. Never claim link OK.
                        mapped := E_NodeState.OFFLINE;
                        linkOk := FALSE;
                    END_IF
                    IF i <= 8 THEN
                        DiagDecodedState[i] := TO_INT(mapped);
                    END_IF
                    IF node >= 1 THEN
                        _pub^.M_SetNodeState(NodeIndex := node, State := mapped, LinkOk := linkOk);
                    END_IF
                END_FOR
                // Couplers/end caps: inferred from the bus answering, never
                // invented. See M_MapPassiveNode.
                FOR i := 1 TO _passiveCount DO
                    IF _passiveNode[i] >= 1 THEN
                        IF reported >= 1 THEN
                            _pub^.M_SetNodeState(NodeIndex := _passiveNode[i],
                                State := E_NodeState.OPERATIONAL, LinkOk := TRUE);
                        ELSE
                            _pub^.M_SetNodeState(NodeIndex := _passiveNode[i],
                                State := E_NodeState.OFFLINE, LinkOk := FALSE);
                        END_IF
                    END_IF
                END_FOR
                // The master node's state is inferred from the read: it answered
                // ADS, so it is running. (A dedicated FB_EcGetMasterState read was
                // dropped to avoid a version-sensitive member name.)
                IF _masterNode >= 1 THEN
                    _pub^.M_SetNodeState(NodeIndex := _masterNode,
                        State := E_NodeState.OPERATIONAL, LinkOk := TRUE);
                END_IF
            ELSE
                // Master unreachable: mark the whole segment (and master) offline.
                _M_PublishAllOffline();
            END_IF
            _firstScanDone := TRUE;
            _step := 20;
        END_IF
    20:
        _tPoll(IN := TRUE, PT := T#250MS);
        IF _tPoll.Q THEN
            _tPoll(IN := FALSE);
            _step := 0;
        END_IF
END_CASE
END_METHOD

// TRUE when the fieldbus is delivering a valid process image: the master read
// succeeded and every slave THE MASTER REPORTS is OPERATIONAL. This is the
// library-detected replacement for a project-declared "bus valid" flag —
// projects no longer wire their own RealBusOk. Derived from the last M_Refresh
// cycle (no extra I/O).
//
// A catalog that declares MORE nodes than are fitted does not make this FALSE:
// per N54 D2 the criterion is that the running bus is functioning properly, and
// a stale catalog is a commissioning issue reported through CountMismatch /
// MappingValid (§10.5.1). Conflating the two silently blocks Control On.
METHOD M_BusOk : BOOL
VAR
    i : INT;
    reported : INT;   // slaves the master actually returned
END_VAR
// N54 D2 (Control On add-on): EnableControlOn is set when the fieldbus masters
// are "functioning properly" — i.e. the bus that is RUNNING is healthy. That is
// deliberately NOT the same question as "does the project catalog list exactly
// the nodes that are fitted": a catalog with more entries than hardware is a
// commissioning/mapping issue (surfaced as CountMismatch and MappingValid,
// §10.5.1), not a running-bus fault, and must not hold off Control On.
M_BusOk := FALSE;
IF NOT _attached OR _fbStates.bError OR NOT ReadOk THEN
    RETURN;  // master unreachable / read failed -> not "functioning properly"
END_IF
// Judge only what the master actually reports. reported = 0 means no slaves on
// the bus at all, which is not a healthy running fieldbus.
reported := TO_INT(_fbStates.nSlaves);
IF reported < 1 THEN
    RETURN;
END_IF
IF reported > _slaveCount THEN
    reported := _slaveCount;   // never read past the mapped buffer
END_IF
FOR i := 1 TO reported DO
    // Zero-based buffer (see _stateBuf): slave i is at i-1. Fully operational iff
    // deviceState is exactly OP (no AL flag bits set).
    IF _stateBuf[i - 1].deviceState <> Tc2_EtherCAT.EC_DEVICE_STATE_OP THEN
        RETURN;  // a slave that IS on the bus is not OP -> bus not valid
    END_IF
END_FOR
// The per-slave read above is refreshed only on demand; the master's own summary
// is sampled every second, so a slave that drops out later is seen here.
IF NOT MasterHealthy THEN
    RETURN;
END_IF
M_BusOk := TRUE;
END_METHOD

// Record one complete master sample; _M_SampleMaster calls it after reading the
// device state, frame statistics and slave CRC counters, and it is the seam a
// fixture drives. The master's counters are cumulative, so each published count
// is the larger of the current window's and the last full window's increase: a
// burst is held for a whole window and a startup's losses never count.
METHOD M_ApplyMasterSample : BOOL
VAR_INPUT
    Ok         : BOOL;      // every read of this sample succeeded
    DevState   : WORD;
    LostFrames : UDINT;     // cumulative lost cyclic + queued frames
    CrcErrors  : UDINT;     // cumulative slave CRC errors, summed over slaves
    MonoNow    : TIME;
END_VAR
VAR
    lostNow : UDINT;
    crcNow : UDINT;
END_VAR
IF Ok THEN
    MasterDevState := DevState;
    IF NOT _mBaselined THEN
        _mLostBase := LostFrames;
        _mCrcBase := CrcErrors;
        _mLastWindowLost := 0;
        _mLastWindowCrc := 0;
        _mWindowStart := MonoNow;
        _mBaselined := TRUE;
    END_IF
    // A counter cleared since the window began counts again from zero.
    IF LostFrames < _mLostBase THEN
        _mLostBase := 0;
    END_IF
    IF CrcErrors < _mCrcBase THEN
        _mCrcBase := 0;
    END_IF
    lostNow := LostFrames - _mLostBase;
    crcNow := CrcErrors - _mCrcBase;
    LostFrameCount := MAX(_mLastWindowLost, lostNow);
    SlaveErrorCount := MAX(_mLastWindowCrc, crcNow);
    IF MonoNow - _mWindowStart >= MASTER_WINDOW THEN
        _mLastWindowLost := lostNow;
        _mLastWindowCrc := crcNow;
        _mLostBase := LostFrames;
        _mCrcBase := CrcErrors;
        _mWindowStart := MonoNow;
    END_IF
    _mSampled := TRUE;
    _mSampledAt := MonoNow;
END_IF
_M_PublishMaster(MonoNow := MonoNow);
M_ApplyMasterSample := Ok;
END_METHOD

METHOD PRIVATE _M_PublishMaster
VAR_INPUT
    MonoNow : TIME;
END_VAR
MasterAvailable := _mSampled AND (MonoNow - _mSampledAt <= MASTER_FRESH_FOR);
MasterHealthy := MasterAvailable AND ((MasterDevState AND MASTER_FAULT_BITS) = 0);
DcSynchronized := MasterAvailable AND ((MasterDevState AND MASTER_DC_NOT_IN_SYNC) = 0);
END_METHOD

// One bounded ADS read at a time: device state, frame statistics, then the slave
// CRC counters; a sample counts only when all three succeeded.
METHOD PRIVATE _M_SampleMaster
VAR
    crc : UDINT;
    n : INT;
    i : INT;
END_VAR
CASE _mPhase OF
    0:
        IF NOT NetIdMissing THEN
            _fbDevState(bExecute := FALSE);
            _fbDevState(sNetId := _netId, bExecute := TRUE, tTimeout := T#1S);
            _mPhase := 1;
        END_IF
    1:
        _fbDevState(bExecute := FALSE);
        IF NOT _fbDevState.bBusy THEN
            IF _fbDevState.bError THEN
                MasterErrorId := _fbDevState.nErrId;
                _mPhase := 9;
            ELSE
                _fbFrames(bExecute := FALSE);
                _fbFrames(sNetId := _netId, bExecute := TRUE, tTimeout := T#1S);
                _mPhase := 2;
            END_IF
        END_IF
    2:
        _fbFrames(bExecute := FALSE);
        IF NOT _fbFrames.bBusy THEN
            IF _fbFrames.bError THEN
                MasterErrorId := _fbFrames.nErrId;
                _mPhase := 9;
            ELSE
                _fbCrc(bExecute := FALSE);
                _fbCrc(sNetId := _netId, pCrcErrorBuf := ADR(_crcBuf),
                    cbBufLen := SIZEOF(_crcBuf), bExecute := TRUE, tTimeout := T#1S);
                _mPhase := 3;
            END_IF
        END_IF
    3:
        _fbCrc(bExecute := FALSE);
        IF NOT _fbCrc.bBusy THEN
            IF _fbCrc.bError THEN
                MasterErrorId := _fbCrc.nErrId;
            ELSE
                // pCrcErrorBuf is zero-based like pStateBuf: slave i is entry i-1.
                crc := 0;
                n := MIN(UINT_TO_INT(_fbCrc.nSlaves), PL_Fraktal.MAX_BUS_NODES + 1);
                FOR i := 0 TO n - 1 DO
                    crc := crc + DWORD_TO_UDINT(_crcBuf[i]);
                END_FOR
                MasterErrorId := 0;
                M_ApplyMasterSample(Ok := TRUE, DevState := _fbDevState.nDevState,
                    LostFrames := _fbFrames.nLostFrames + _fbFrames.nLostQueuedFrames,
                    CrcErrors := crc, MonoNow := TIME());
            END_IF
            _mPhase := 9;
        END_IF
    9:
        _mPoll(IN := TRUE, PT := MASTER_POLL);
        IF _mPoll.Q THEN
            _mPoll(IN := FALSE, PT := MASTER_POLL);
            _mPhase := 0;
        END_IF
ELSE
    _mPhase := 0;
END_CASE
_M_PublishMaster(MonoNow := TIME());   // freshness expires even while a read hangs
END_METHOD

// §10.5.1 demand gate. Call every cycle with Active := TRUE while a consumer is
// reading the bus picture (the HMI fieldbus view is open, or a mailbox scan was
// requested); FALSE parks the scanner. Held states are NOT invalidated on
// release — a stale-but-true picture beats a fabricated one; the view re-reads
// on its next activation.
METHOD M_RequestScan
VAR_INPUT
    Active : BOOL;
END_VAR
IF Active AND NOT _scanRequested THEN
    // Re-arm immediately on a rising request so opening the view does not wait
    // out the poll timer.
    _tPoll(IN := FALSE);
    IF _step = 20 THEN
        _step := 0;
    END_IF
END_IF
_scanRequested := Active;
END_METHOD

// Fail-visible fallback: publish every mapped node (and the master) as OFFLINE.
// Used when the master cannot be reached and when its AmsNetId cannot be
// resolved -- an unknown bus must never look "operational" on the HMI.
METHOD PRIVATE _M_PublishAllOffline
VAR
    i : INT;
    node : INT;
END_VAR
IF NOT _attached THEN
    RETURN;
END_IF
FOR i := 1 TO _slaveCount DO
    node := _slaveNode[i];
    IF node >= 1 THEN
        _pub^.M_SetNodeState(NodeIndex := node,
            State := E_NodeState.OFFLINE, LinkOk := FALSE);
    END_IF
END_FOR
// Couplers/end caps go dark with the bus they carry.
FOR i := 1 TO _passiveCount DO
    IF _passiveNode[i] >= 1 THEN
        _pub^.M_SetNodeState(NodeIndex := _passiveNode[i],
            State := E_NodeState.OFFLINE, LinkOk := FALSE);
    END_IF
END_FOR
IF _masterNode >= 1 THEN
    _pub^.M_SetNodeState(NodeIndex := _masterNode,
        State := E_NodeState.OFFLINE, LinkOk := FALSE);
END_IF
END_METHOD

// Decode an ST_EcSlaveState.deviceState byte (Beckhoff Tc2_EtherCAT, EtherCAT
// AL state machine) into the neutral E_NodeState the HMI renders.
//   low nibble  = AL state: INIT=1, PREOP=2, BOOTSTRAP=3, SAFEOP=4, OP=8
//   high nibble = flags:    ERROR=0x10, INVALID_VPRS=0x20, INITCMD_ERROR=0x40,
//                           DISABLED=0x80  -> any set is a fault.
// Source: infosys.beckhoff.com ST_EcSlaveState / EC_DEVICE_STATE_*.
METHOD PRIVATE _M_MapSlaveState : E_NodeState
VAR_INPUT
    DeviceState : BYTE;
END_VAR
// Any diagnostic flag bit (high nibble) overrides the AL state -> FAULT.
// After that check only the AL-state bits remain, so compare directly.
IF (DeviceState AND 16#F0) <> 0 THEN
    _M_MapSlaveState := E_NodeState.FAULT;
ELSIF DeviceState = Tc2_EtherCAT.EC_DEVICE_STATE_OP THEN
    _M_MapSlaveState := E_NodeState.OPERATIONAL;
ELSIF DeviceState = Tc2_EtherCAT.EC_DEVICE_STATE_SAFEOP THEN
    _M_MapSlaveState := E_NodeState.SAFEOP;
ELSIF DeviceState = Tc2_EtherCAT.EC_DEVICE_STATE_PREOP THEN
    _M_MapSlaveState := E_NodeState.PREOP;
ELSIF DeviceState = Tc2_EtherCAT.EC_DEVICE_STATE_INIT THEN
    _M_MapSlaveState := E_NodeState.INIT;
ELSE
    // BOOTSTRAP (0x03) or no state reported -> show as offline.
    _M_MapSlaveState := E_NodeState.OFFLINE;
END_IF
END_METHOD

END_FUNCTION_BLOCK

// ---- Connectivity/FB_IoTopologyPublisher.TcPOU
// Core §10.5.1 infrastructure service. Owns the reusable bounded-table,
// validation, health and diagnostic-join algorithms; project code supplies only
// physical topology metadata and live values. This is not a module tier.
FUNCTION_BLOCK FB_IoTopologyPublisher
VAR
    {attribute 'OPC.UA.DA' := '0'}
    _data : REFERENCE TO ST_FieldbusTopology;
    _attached : BOOL;
END_VAR

;

METHOD Setup : BOOL
VAR_INPUT
    DataRef : REFERENCE TO ST_FieldbusTopology;
    ResetData : BOOL;
END_VAR
VAR
    n, c : INT;
END_VAR
_data REF= DataRef;
_attached := __ISVALIDREF(_data);
IF _attached AND ResetData THEN
    _data.NodeCount := 0;
    _data.MappingValid := TRUE;
    _data.MappingDiagnostic := '';
    FOR n := 1 TO PL_Fraktal.MAX_BUS_NODES DO
        _data.Nodes[n].Name := '';
        _data.Nodes[n].DescriptionKey := '';
        _data.Nodes[n].TypeId := '';
        _data.Nodes[n].Address := '';
        _data.Nodes[n].ParentIdx := 0;
        _data.Nodes[n].ChannelCount := 0;
        FOR c := 1 TO PL_Fraktal.MAX_NODE_CHANNELS DO
            _data.Nodes[n].Channels[c].Name := '';
            _data.Nodes[n].Channels[c].Path := '';
        END_FOR
    END_FOR
ELSIF _attached THEN
    ;
ELSE
    _attached := FALSE;
END_IF
Setup := _attached;
END_METHOD

